// SIMATIC S7-200 SMART project (STEP 7-Micro/WIN SMART), CPU SR40

SYMBOL_TABLE 表格 1
Stage1_Temp_CT   C0       // 阶段升温一计数器，分钟计数
Stage2_Temp_CT   C1       // 阶段升温二计数器，分钟计数
Stage3_Temp_CT   C2       // 阶段升温三计数器，分钟计数
Stage4_Temp_CT   C3       // 阶段升温四计数器，分钟计数
Stage5_Temp_CT   C4       // 阶段升温五计数器，分钟计数
Stage6_Temp_CT   C5       // 阶段升温六计数器，分钟计数
Sys_Time_Minutes_CNT C100     // 系统运行时长计数器，分钟
Sys_Time_Hours_CNT C101     // 系统运行时长计数器，小时
Sys_Time_Repeat_CNT C102     // 系统运行时长轮数计数器，超过32767小时后，该轮数加1，小时归0
C_Leak_CountDown_CT C103     // 检漏倒计时 计数器
C_Valve_Detect_CT C104     // 调节阀检测倒计时 计数器
C_Purge_CountDown_CT C105     // 吹扫倒计时 计数器
C_Ignite_CountDown_CT C106     // 点火 倒计时 计数器
MBUS_INIT_DONE   M0.1     // MBUS_INIT的Done 状态位
MBUS_SLAVE_DONE  M0.2     // MBUS_SLAVE Done状态位
M_Safety_Check_FLG M0.3     // 系统安全回路检测 标志，如压力、检漏、前火检等
M_Valve_ALM_FLG  M0.4     // 调节阀检测故障标志
M_Local_Remote_FLG M0.5     // 本地远程标志，1本地，0远程
M_Auto_Temp_FLG  M0.6     // 自动升温控制标志
M_Purge_Display_FLG M0.7     // 显示吹扫动画
M_SYS_Safety_Pass_FLG M1.0     // 安全自检通过标志：检漏通过、空气压力正常、燃气压力正常，前火检正常
M_Sys_Run_FLG    M1.1     // 启动标志
M_Purge_Begin_FLG M1.2     // 开始吹扫标志
M_Ignite_Begin_FLG M1.3     // 开始点火标志
M_Ignite_Success_FLG M1.4     // 点火成功标志
M_OverTemp_FLG   M1.5     // 超温标志
M_Purge_Finish_FLG M1.6     // 吹扫结束标志
M_Ignite_Ready_FLG M1.7     // 点火准备标志
M_SYS_Alarm_FLG  M2.0     // 系统故障标志
M_Ignite_BeginTime_FLG M2.1     // 点火延时开始
M_Temp1_Read_FLG M2.2     // 读阶段1温度标志
M_Temp2_Read_FLG M2.3     // 读阶段2温度标志
M_Temp3_Read_FLG M2.4     // 读阶段3温度标志
M_Temp4_Read_FLG M2.5     // 读阶段4温度标志
M_Temp5_Read_FLG M2.6     // 读阶段5温度标志
M_Temp6_Read_FLG M2.7     // 读阶段6温度标志
M_Valve_Pass_FLG M3.0     // 调节阀检测通过标志
M_Leak_Exception_FLG M3.1     // 检漏异常报警
M_Leak_Pass_FLG  M3.4     // 检漏程序，检漏通过
M_Run_Big_Fire_FLG M3.5     // 大火指示，表示大火正常燃烧
M_TA_Spark_FLG   M3.7     // 变压器打火标志
M_Temp_Error_FLG M4.0     // 温度错误，DCS传送温度数据有误，请
M_Valve_Ignite_OPEN_FLG M4.1     // 点火阀开启标志
M_Sys_Detect_PASS_FLG M4.2     // 系统预检通过标志
Local_Start_CMD  M10.0    // 本地启动指令
Local_Stop_CMD   M10.1    // 本地停止指令
Local_Reset_CMD  M10.2    // 本地复位指令
Remote_Start_CMD M10.3    // 远程启动指令
Remote_Stop_CMD  M10.4    // 远程停止指令
Remote_Reset_CMD M10.5    // 远程复位指令
M_Manu_TurnUp_CMD M10.6    // 手动升档，触摸屏虚拟按钮
M_Manu_TurnDown_CMD M10.7    // 手动降档，触摸屏虚拟按钮
M_Auto_Manu_CMD  M11.0    // 自动/手动切换，触摸屏虚拟按钮，1自动，0手动
M_Leak_ValveCut_CMD M11.1    // 检漏程序，打开主火阀（切断阀）指令
M_ValveCut_CMD   M11.2    // 主程序，打开主火阀（切断阀）
M_Leak_ValveSafety_CMD M11.3    // 检漏程序，打开安全阀 指令
M_ValveSafety_CMD M11.4    // 主程序，打开安全阀 指令
Remote_TurnUP_CMD M11.5    // 远程升档指令
Remote_TurnDown_CMD M11.6    // 远程降档指令
Local_TurnUP_CMD M11.7    // 本地升档指令
Local_TurnDown_CMD M12.0    // 本地降档指令
M_Leak_Start_CMD M12.1    // 手动检漏 虚拟按钮
M_Valve_Detect_CMD M12.2    // 手动调节阀检测 虚拟按钮
M_Ignite_Failed_ALM M20.0    // 点火失败报警
M_Flame_Loss_ALM M20.1    // 火焰信号丢失
M_DCS_Lock_ALM   M20.2    // DCS安全联锁故障
M_Air_Pres_Low_ALM M20.3    // 空气压力低故障
M_Gas_Pres_High_ALM M20.4    // 燃气压力高故障
M_Gas_Pres_Low_ALM M20.5    // 燃气压力低故障
M_Flame_Pre_ALM  M20.6    // 点火前发现火焰故障
M_Leak_Exception2_ALM M20.7    // 检漏程序，第2步检漏异常标志
M_Leak_Exception4_ALM M21.0    // 检漏程序，第4步检漏异常标志
M_Valve_Air_ALM  M21.1    // 空气调节阀故障
M_Valve_Gas_ALM  M21.2    // 燃气调节阀故障
T_Purge_Duration T101     // 吹扫时长定时器
T_Ignite_Delay   T102     // 点火延时定时器，从调节阀走到位到高压包放电之间的时间间隔
T_Level_Interval T103     // 升降档间隔定时器
T_Flame_Loss_Delay T104     // 火焰丢失延时定时器
T_VAL_Open_Delay T105     // 大火阀开启延时定时器
T_TA_Spark_Time  T106     // 高压包打火时长定时器
T_Valve_Ignite_Delay T107     // 母火阀延时打开定时器
T_Leak_Step1_Delay T110     // 检漏第1步延时定时器
T_Leak_Step2_Delay T111     // 检漏第2步延时定时器
T_Leak_Step3_Delay T112     // 检漏第3步延时定时器
T_Leak_Step4_Delay T113     // 检漏第4步延时定时器
T_Valve_Control_Detect T115     // 调节阀检测定时器
T_Ignite_ValveGo_Delay T116     // 点火位置，调节阀走至点火位置延时
T_Flame_Pre_Detect T118     // 前火焰检测延时定时器
T_Purge_ValveOpenDelay T119     // 吹扫 调节阀开启延时定时器
T_Flame_Build_Delay T120     // 火焰建立延时定时器
T_Leak_Total_Time T121     // 检漏总时长定时器
I_DCS_Abandon    V0.0     // I_DCS安全联锁，不用
I_Air_Pres_Low_STS V0.1     // 空气压力低故障
I_Gas_Pres_High_STS V0.2     // 燃气压力高故障
I_Gas_Pres_Low_STS V0.3     // 燃气压力低故障
I_JES258_Alrm_Abandon V0.4     // I_JES258故障不用
I_Flame_STS      V0.5     // 火焰信号
I_Run_STS        V0.6     // 启动按钮信号
I_Stop_STS       V0.7     // 停止按钮信号
I_Reset_STS      V1.0     // 复位按钮信号
I_LocalRemote_STS V1.1     // 本地、远程信号。1本地、0远程
Q_Sys_Alarm      V2.0     // 系统报警输出指令，蜂鸣器
Q_Valve_Ignite   V2.1     // 点火阀Ignite打开命令
Q_Valve_Cut      V2.2     // 主火切断阀打开命令
Q_TA_Spark       V2.3     // 变压器打火指令
Q_SYS_Flame_Light V2.4     // 有火指示灯
Q_SYS_Run_Light  V2.5     // 运行指示灯
Q_SYS_Stop_Light V2.6     // 停止指示灯
Q_Valve_Safety   V2.7     // 安全阀打开命令
V_Remote_Alarm_Status V1620.0  // 故障状态RTU
V_Remote_Auto_Status V1620.1  // 自动状态RTU
V_Remote_Run_Status V1620.2  // 启动状态RTU
V_Remote_Stop_Status V1620.3  // 停止状态RTU
V_Local_Remote_Status V1620.4  // 本地远程状态RTU
V_Remote_Run_CMD V1620.5  // 远程启动RTU
V_Remote_Stop_CMD V1620.6  // 远程停止RTU
V_Remote_Reset_CMD V1620.7  // 远程复位RTU
V_Remote_TurnUp_CMD V1621.0  // 远程升档RTU
V_Remote_TurnDown_CMD V1621.1  // 远程降档RTU
V_PID_ErrorCode  VB800    // PID 控制错误码
V_MBUS_INIT_Error VB802    // MBUS_INIT Error 错误码
V_MBUS_SLAVE_Error VB804    // MBUS_SLAVE Error 错误码
B_Leak_Step_Num  VB806    // 检漏步数，第1、2、3、4步
B_Leak_Status    VB808    // 检漏状态，0:停止检漏 1:检漏中 2:检漏完成
B_ValveLift_Status VB810    // 调节阀检测状态，0停止检测、1检测中、2检测完成
B_Ignate_Backup_Status VB812    // 0正常；1点火备用，取消前火检
DI_Current_Temp_VAL VD20     // 当前温度（长整型）数据来自DCS
R_Current_Temp_Display VD24     // 温度HMI显示值
R_ValveLift_Gas_VAL_Per VD32     // 燃气阀门开度显示%
R_ValveLift_Air_VAL_Per VD36     // 空气阀门开度显示%
R_Valve_Gas_DIFF_ABS VD40     // 燃气阀门给定值与反馈值之差，取绝对值
R_Valve_Air_DIFF_ABS VD44     // 空气阀门给定值与反馈值之差，取绝对值
R_ValveLift_Gas_VAL VD48     // 当前燃气给定值
R_ValveLift_Air_VAL VD52     // 当前空气给定值
R_PID_Temp_VAL   VD56     // PID当前目标温度
R_PID_Manu_VAL   VD60     // PID手动值
R_Purge_BeginTime_VAL VD64     // 吹扫计时开始_值
R_PID_Level_Round_VAL VD68     // PID输出换算成档位，四舍五入后
R_Current_Level_VAL VD72     // 当前档位值
R_PID_EachLevel_VAL VD76     // 当量_每档
R_PID_Output_VAL VD80     // 转换为实数后的PID输出值
R_PID_Level_VAL  VD84     // PID输出换算成档位
R_Current_Temp_VAL VD88     // 当前温度（实数）数据来自DCS
R_Valve_Gas_DIFF_VAL VD92     // 燃气阀门给定值与反馈值之差
R_Valve_Air_DIFF_VAL VD96     // 空气阀门给定值与反馈值之差
DI_ValveLift_Air_Per VD148    // 空气调节阀 双整型 %
DI_ValveLift_Gas_Per VD156    // 燃气调节阀 双整型 %
R_Temp_Upper_Limit_SET VD300    // 温度上限设定值
R_Temp_Lower_Limit_SET VD304    // 温度下限设定值
R_Over_Temp_Stop_SET VD308    // 超温停机设定值
R_Gas_DiffAlow_SET VD312    // 燃气偏差允许值设定
R_Air_DiffAlow_SET VD316    // 空气偏差允许值设定
R_Purge_Valve_Air_SET VD320    // 吹扫空气阀开度设定值
R_PID_D_SET      VD324    // PID微分_D 设定值
R_PID_P_SET      VD328    // PID增益_P 设定值
R_PID_I_SET      VD332    // PID积分_I 设定值
R_PID_Ts_SET     VD336    // PID采样时间设定值
R_Level_Total_SET VD340    // 档位设置
R_Gas_Level_Stop_SET VD344    // 燃气停机档设定值
R_Gas_Level_Ignite_SET VD348    // 燃气点火档设定值
R_Gas_Level1_SET VD352    // 燃气1档设定值
R_Gas_Level2_SET VD356    // 燃气2档设定值
R_Gas_Level3_SET VD360    // 燃气3档设定值
R_Gas_Level4_SET VD364    // 燃气4档设定值
R_Gas_Level5_SET VD368    // 燃气5档设定值
R_Gas_Level6_SET VD372    // 燃气6档设定值
R_Gas_Level7_SET VD376    // 燃气7档设定值
R_Gas_Level8_SET VD380    // 燃气8档设定值
R_Gas_Level9_SET VD384    // 燃气9档设定值
R_Gas_Level10_SET VD388    // 燃气10档设定值
R_Gas_Level11_SET VD392    // 燃气11档设定值
R_Gas_Level12_SET VD396    // 燃气12档设定值
R_Gas_Level13_SET VD400    // 燃气13档设定值
R_Gas_Level14_SET VD404    // 燃气14档设定值
R_Gas_Level15_SET VD408    // 燃气15档设定值
R_Gas_Level16_SET VD412    // 燃气16档设定值
R_Gas_Level17_SET VD416    // 燃气17档设定值
R_Gas_Level18_SET VD420    // 燃气18档设定值
R_Air_Level_Stop_SET VD424    // 空气停机档设定值
R_Air_Level_Ignite_SET VD428    // 空气点火档设定值
R_Air_Level1_SET VD432    // 空气1档设定值
R_Air_Level2_SET VD436    // 空气2档设定值
R_Air_Level3_SET VD440    // 空气3档设定值
R_Air_Level4_SET VD444    // 空气4档设定值
R_Air_Level5_SET VD448    // 空气5档设定值
R_Air_Level6_SET VD452    // 空气6档设定值
R_Air_Level7_SET VD456    // 空气7档设定值
R_Air_Level8_SET VD460    // 空气8档设定值
R_Air_Level9_SET VD464    // 空气9档设定值
R_Air_Level10_SET VD468    // 空气10档设定值
R_Air_Level11_SET VD472    // 空气11档设定值
R_Air_Level12_SET VD476    // 空气12档设定值
R_Air_Level13_SET VD480    // 空气13档设定值
R_Air_Level14_SET VD484    // 空气14档设定值
R_Air_Level15_SET VD488    // 空气15档设定值
R_Air_Level16_SET VD492    // 空气16档设定值
R_Air_Level17_SET VD496    // 空气17档设定值
R_Air_Level18_SET VD500    // 空气18档设定值
R_Stage1_Temp_SET VD504    // 阶段1温度设定值
R_Stage2_Temp_SET VD508    // 阶段2温度设定值
R_Stage3_Temp_SET VD512    // 阶段3温度设定值
R_Stage4_Temp_SET VD516    // 阶段4温度设定值
R_Stage5_Temp_SET VD520    // 阶段5温度设定值
R_Stage6_Temp_SET VD524    // 阶段6温度设定值
R_Remote_AirLift_VAL VD640    // 远程显示空气阀开度
R_Remote_GasLift_VAL VD644    // 远程显示燃气阀开度
R_Remote_Temp_VAL VD648    // 远程显示温度
R_Remote_Air_VAL VD1640   // 空气调节阀开度RTU
R_Remote_Gas_VAL VD1644   // 燃气调节阀开度RTU
R_Remote_Level_VAL VD1652   // 当前档位RTU
R_Remote_Temp_SET VD1880   // 目标温度RTU
W_Purge_Time_VAL VW100    // 当前吹扫时长显示值
W_PID_Output_VAL VW104    // PID输出
W_Stage1_Temp_Time_VAL VW108    // 第1阶段温度保持时长显示，分钟
W_Stage2_Temp_Time_VAL VW112    // 第2阶段温度保持时长显示，分钟
W_Stage3_Temp_Time_VAL VW116    // 第3阶段温度保持时长显示，分钟
W_Stage4_Temp_Time_VAL VW120    // 第4阶段温度保持时长显示，分钟
W_Stage5_Temp_Time_VAL VW124    // 第5阶段温度保持时长显示，分钟
W_Stage6_Temp_Time_VAL VW128    // 第6阶段温度保持时长显示，分钟
W_Sys_Time_Hour_VAL VW132    // HMI显示运行小时
W_Sys_Time_Minute_VAL VW136    // HMI显示运行分钟
W_Valve_Detect_CD_VAL VW138    // 调节阀检测倒计时 计算值
W_Leak_CD_VAL    VW140    // 检漏倒计时 计算值
W_Purge_CD_VAL   VW142    // 吹扫倒计时 计算值
W_Ignite_CD_VAL  VW144    // 高压打火 倒计时 计算值
W_ValveLift_Air_VAL_Per VW152    // 空气调节阀开度 整数 %
W_ValveLift_Gas_VAL_Per VW158    // 燃气调节阀开度 整数 %
W_Purge_Time_SET VW528    // 吹扫时间设定
W_Ignite_Delay_SET VW532    // 点火延时设定值
W_ValveCut_Delay_SET VW536    // 主火阀(切断阀)开启延时设定值
W_Stage1_Temp_Time_SET VW540    // 第1阶段温度时长设定值，小时
W_Stage2_Temp_Time_SET VW544    // 第2阶段温度时长设定值，小时
W_Stage3_Temp_Time_SET VW548    // 第3阶段温度时长设定值，小时
W_Stage4_Temp_Time_SET VW552    // 第4阶段温度时长设定值，小时
W_Stage5_Temp_Time_SET VW556    // 第5阶段温度时长设定值，小时
W_Stage6_Temp_Time_SET VW560    // 第6阶段温度时长设定值，小时
W_PreFlame_Time_SET VW564    // 前火检时长设定值
W_Ignite_Spark_Time_SET VW568    // 高压包打火时长设定值
W_Valve_Ignite_Time_SET VW572    // 点火阀开启延时设定值
W_ValveDetect_Time_SET VW576    // 调节阀检测时长设定值
W_Flame_Build_Time_SET VW580    // 火焰建立延时时长设定值
W_Flame_Loss_Time_SET VW584    // 火焰丢失延时时长设定值，建议1~3秒
W_Sys_Status     VW814    // 1.检漏、调节阀检测中…… / 2.检测完成 / 3.设备停止 / 4.正在启动…… / 5.正在吹扫…… / 6.吹扫完成 / 7.点火准备中…… / 8.正在点火…… / 9.点火成功 / 10.【小火运行】 / 11.【大火运行】 / 12.故障报警
W_Sys_Status_Time VW816    // 系统状态时间
W_Remote_Temp_VAL VW1898   // 当前温度RTU
W_Remote_Air_P_VAL VW1918   // 当前管道空气压力，风压
END_SYMBOL_TABLE

SYMBOL_TABLE 系统符号
Always_On        SM0.0    // 始终接通
First_Scan_On    SM0.1    // 仅在第一个扫描周期时接通
Clock_60s        SM0.4    // 针对 1 分钟的周期时间，时钟脉冲接通 30 s，断开 30 s.
Clock_1s         SM0.5    // 针对 1 s 的周期时间，时钟脉冲接通 0.5 s，断开 0.5 s.
END_SYMBOL_TABLE

ORGANIZATION_BLOCK 程序块:OB1
TITLE=程序注释
BEGIN
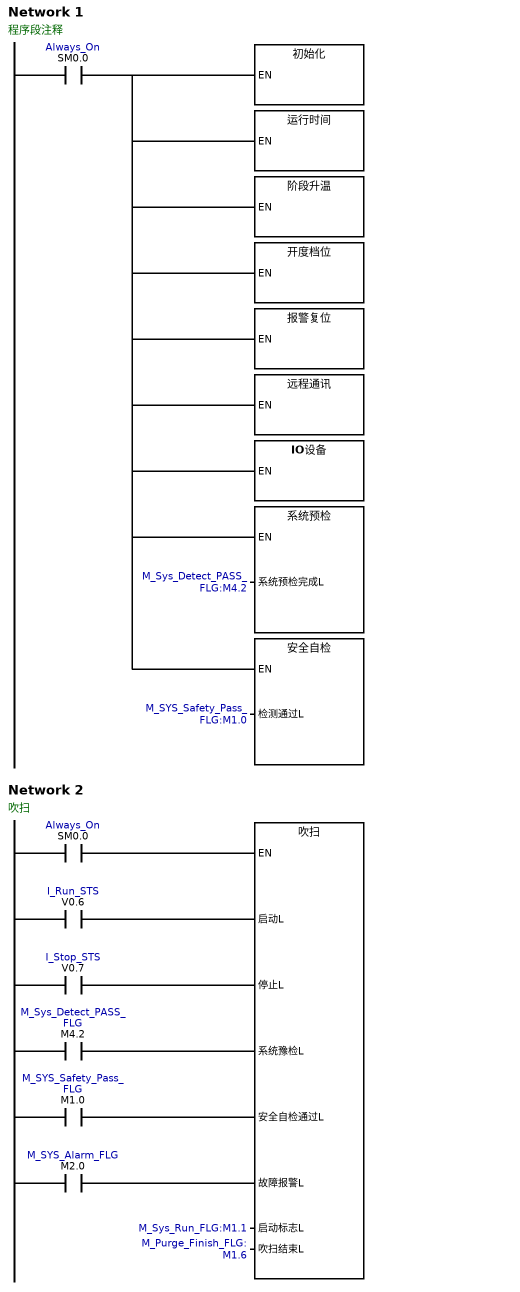
Network 1
// 程序段注释
LD     Always_On:SM0.0
CALL   初始化:SBR0
CALL   运行时间:SBR9
CALL   阶段升温:SBR5
CALL   开度档位:SBR6
CALL   报警复位:SBR13
CALL   远程通讯:SBR7
CALL   IO设备:SBR8
CALL   系统预检:SBR1, M_Sys_Detect_PASS_FLG:M4.2
CALL   安全自检:SBR2, M_SYS_Safety_Pass_FLG:M1.0
Network 2
// 吹扫
LD     Always_On:SM0.0
=      L60.0
LD     I_Run_STS:V0.6
=      L63.7
LD     I_Stop_STS:V0.7
=      L63.6
LD     M_Sys_Detect_PASS_FLG:M4.2
=      L63.5
LD     M_SYS_Safety_Pass_FLG:M1.0
=      L63.4
LD     M_SYS_Alarm_FLG:M2.0
=      L63.3
LD     L60.0
CALL   吹扫:SBR3, L63.7, L63.6, L63.5, L63.4, L63.3, M_Sys_Run_FLG:M1.1, M_Purge_Finish_FLG:M1.6
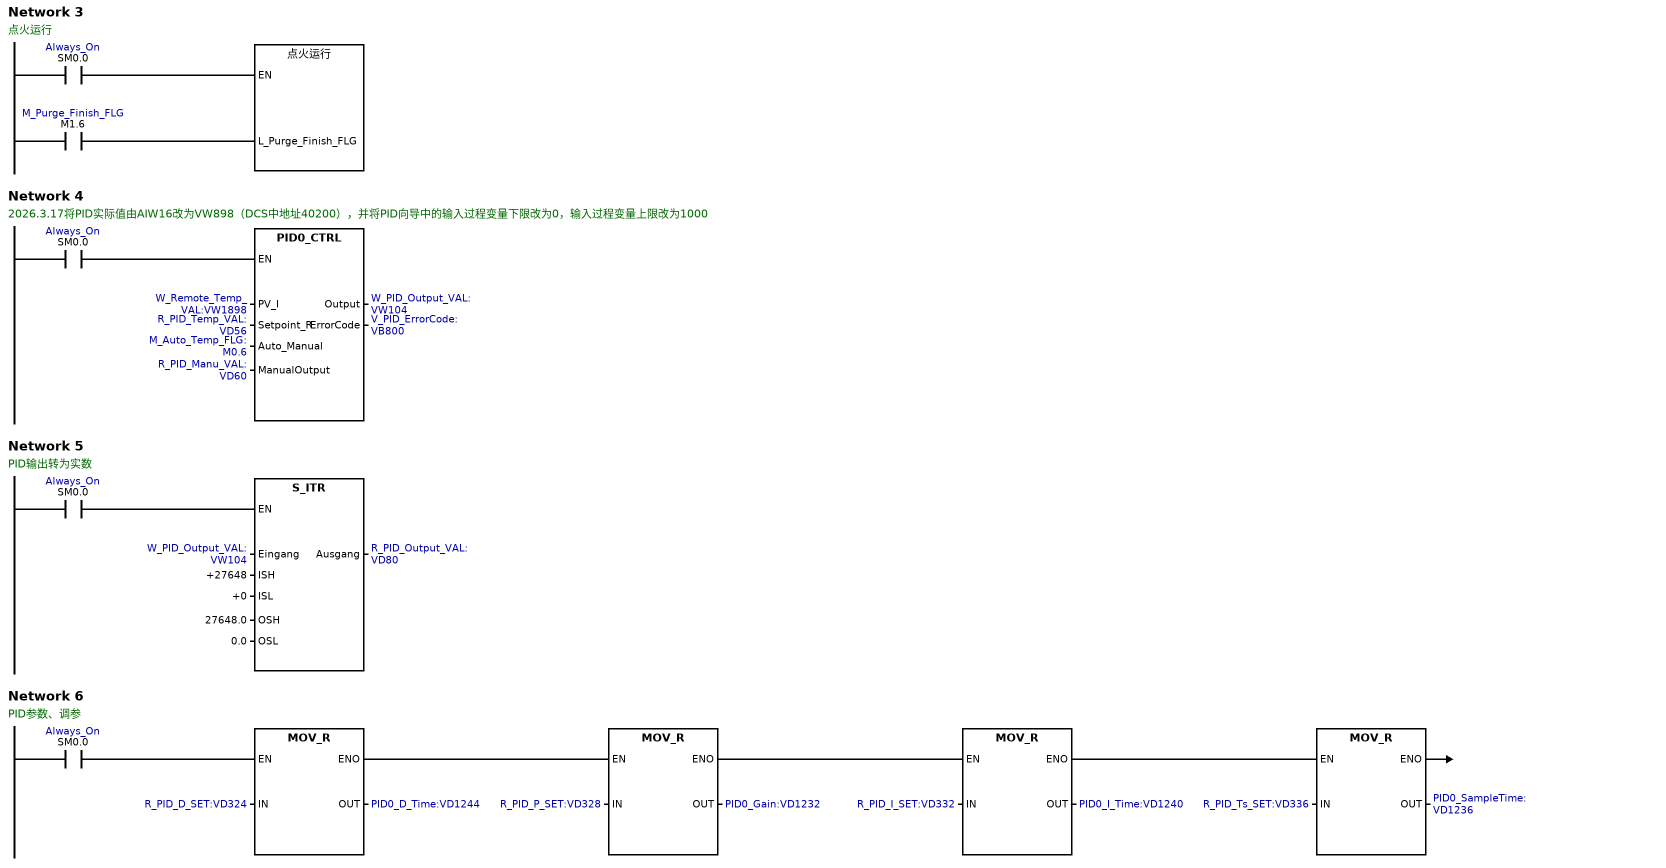
Network 3
// 点火运行
LD     Always_On:SM0.0
=      L60.0
LD     M_Purge_Finish_FLG:M1.6
=      L63.7
LD     L60.0
CALL   点火运行:SBR4, L63.7
Network 4
// 2026.3.17将PID实际值由AIW16改为VW898（DCS中地址40200），并将PID向导中的输入过程变量下限改为0，输入过程变量上限改为1000
LD     Always_On:SM0.0
CALL   PID0_CTRL:SBR18, W_Remote_Temp_VAL:VW1898, R_PID_Temp_VAL:VD56, M_Auto_Temp_FLG:M0.6, R_PID_Manu_VAL:VD60, W_PID_Output_VAL:VW104, V_PID_ErrorCode:VB800
Network 5
// PID输出转为实数
LD     Always_On:SM0.0
CALL   S_ITR:SBR30, W_PID_Output_VAL:VW104, +27648, +0, 27648.0, 0.0, R_PID_Output_VAL:VD80
Network 6
// PID参数、调参
LD     Always_On:SM0.0
MOVR   R_PID_D_SET:VD324, PID0_D_Time:VD1244
AENO
MOVR   R_PID_P_SET:VD328, PID0_Gain:VD1232
AENO
MOVR   R_PID_I_SET:VD332, PID0_I_Time:VD1240
AENO
MOVR   R_PID_Ts_SET:VD336, PID0_SampleTime:VD1236
END_ORGANIZATION_BLOCK

SUBROUTINE_BLOCK 初始化:SBR0
TITLE=初始化子程序
// 功能：数据初始化
// 1、本地/远程转换
// 2、PID自动/手动转换
// 3、PLC IO 输入输出映射
// 4、数据初始化
// 5、本地/远程 命令封装
// 6、模拟量处理
// 
// 
BEGIN
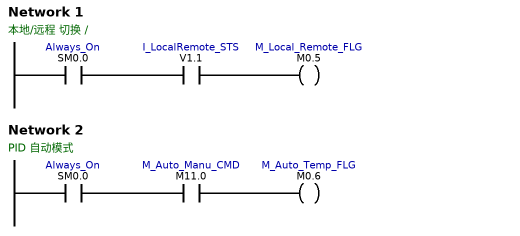
Network 1
// 本地/远程 切换
// 
LD     Always_On:SM0.0
A      I_LocalRemote_STS:V1.1
=      M_Local_Remote_FLG:M0.5
Network 2
// PID 自动模式 
LD     Always_On:SM0.0
A      M_Auto_Manu_CMD:M11.0
=      M_Auto_Temp_FLG:M0.6
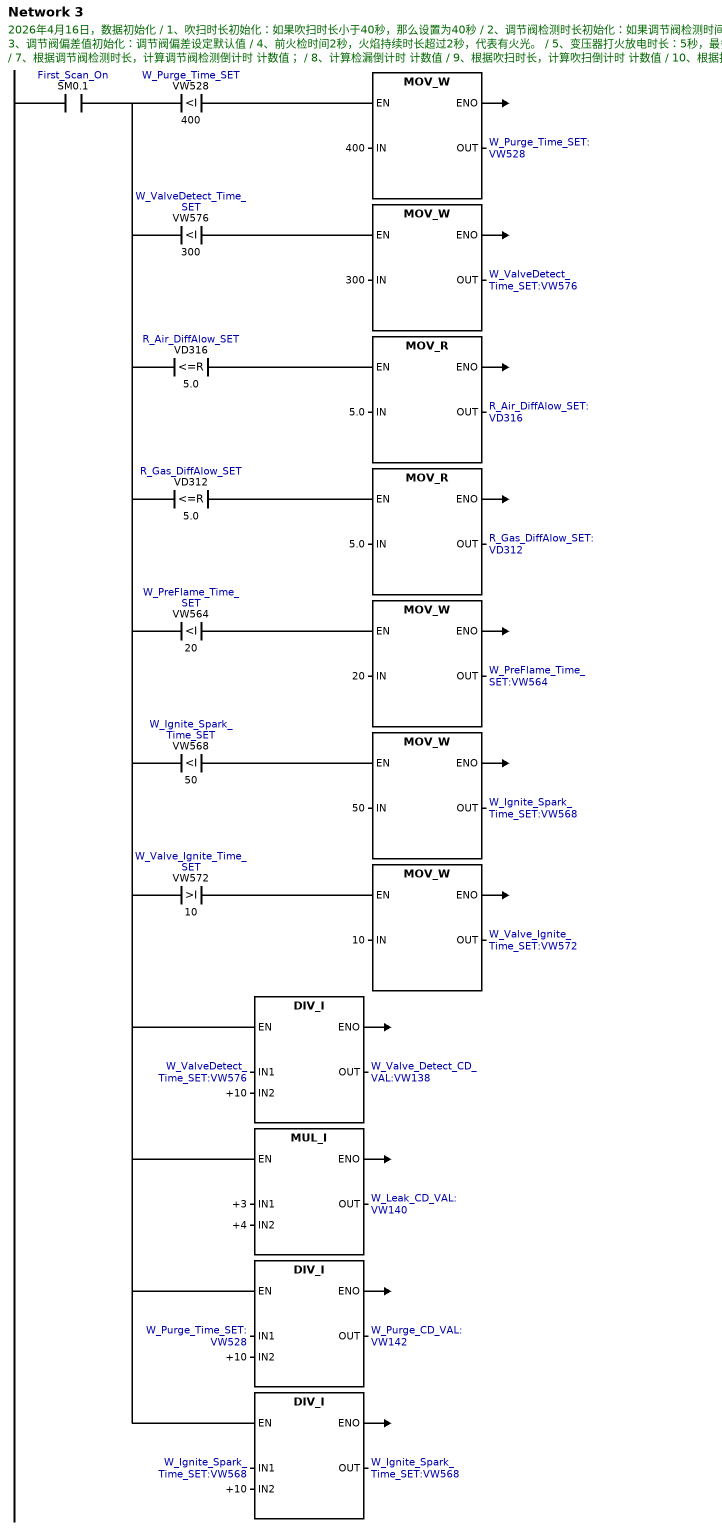
Network 3
// 2026年4月16日，数据初始化
// 1、吹扫时长初始化：如果吹扫时长小于40秒，那么设置为40秒
// 2、调节阀检测时长初始化：如果调节阀检测时间小于30秒，那么设置为30秒
// 3、调节阀偏差值初始化：调节阀偏差设定默认值
// 4、前火检时间2秒，火焰持续时长超过2秒，代表有火光。
// 5、变压器打火放电时长：5秒，最多7秒，大于7秒，那么 就设置为7秒
// 6、点火阀延时开启时长：1秒，最多2秒
// 7、根据调节阀检测时长，计算调节阀检测倒计时 计数值；
// 8、计算检漏倒计时 计数值
// 9、根据吹扫时长，计算吹扫倒计时 计数值
// 10、根据打火时长，计算打火倒计时 计数值
LD     First_Scan_On:SM0.1
LPS
AW<    W_Purge_Time_SET:VW528, 400
MOVW   400, W_Purge_Time_SET:VW528
LRD
AW<    W_ValveDetect_Time_SET:VW576, 300
MOVW   300, W_ValveDetect_Time_SET:VW576
LRD
AR<=   R_Air_DiffAlow_SET:VD316, 5.0
MOVR   5.0, R_Air_DiffAlow_SET:VD316
LRD
AR<=   R_Gas_DiffAlow_SET:VD312, 5.0
MOVR   5.0, R_Gas_DiffAlow_SET:VD312
LRD
AW<    W_PreFlame_Time_SET:VW564, 20
MOVW   20, W_PreFlame_Time_SET:VW564
LRD
AW<    W_Ignite_Spark_Time_SET:VW568, 50
MOVW   50, W_Ignite_Spark_Time_SET:VW568
LRD
AW>    W_Valve_Ignite_Time_SET:VW572, 10
MOVW   10, W_Valve_Ignite_Time_SET:VW572
LRD
MOVW   W_ValveDetect_Time_SET:VW576, W_Valve_Detect_CD_VAL:VW138
/I     +10, W_Valve_Detect_CD_VAL:VW138
LRD
MOVW   +3, W_Leak_CD_VAL:VW140
*I     +4, W_Leak_CD_VAL:VW140
LRD
MOVW   W_Purge_Time_SET:VW528, W_Purge_CD_VAL:VW142
/I     +10, W_Purge_CD_VAL:VW142
LPP
/I     +10, W_Ignite_Spark_Time_SET:VW568
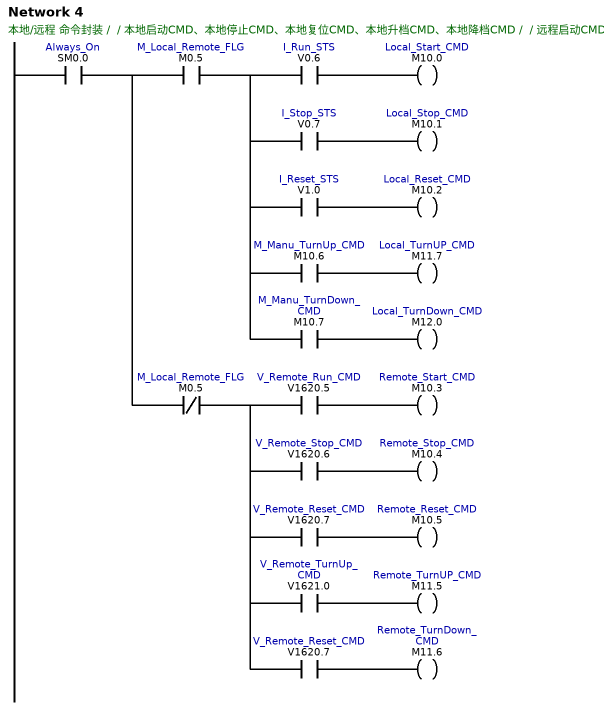
Network 4
// 本地/远程 命令封装
// 
// 本地启动CMD、本地停止CMD、本地复位CMD、本地升档CMD、本地降档CMD
// 
// 远程启动CMD、远程停止CMD、远程复位CMD、远程升档CMD、远程降档CMD
LD     Always_On:SM0.0
LPS
A      M_Local_Remote_FLG:M0.5
LPS
A      I_Run_STS:V0.6
=      Local_Start_CMD:M10.0
LRD
A      I_Stop_STS:V0.7
=      Local_Stop_CMD:M10.1
LRD
A      I_Reset_STS:V1.0
=      Local_Reset_CMD:M10.2
LRD
A      M_Manu_TurnUp_CMD:M10.6
=      Local_TurnUP_CMD:M11.7
LPP
A      M_Manu_TurnDown_CMD:M10.7
=      Local_TurnDown_CMD:M12.0
LPP
AN     M_Local_Remote_FLG:M0.5
LPS
A      V_Remote_Run_CMD:V1620.5
=      Remote_Start_CMD:M10.3
LRD
A      V_Remote_Stop_CMD:V1620.6
=      Remote_Stop_CMD:M10.4
LRD
A      V_Remote_Reset_CMD:V1620.7
=      Remote_Reset_CMD:M10.5
LRD
A      V_Remote_TurnUp_CMD:V1621.0
=      Remote_TurnUP_CMD:M11.5
LPP
A      V_Remote_Reset_CMD:V1620.7
=      Remote_TurnDown_CMD:M11.6
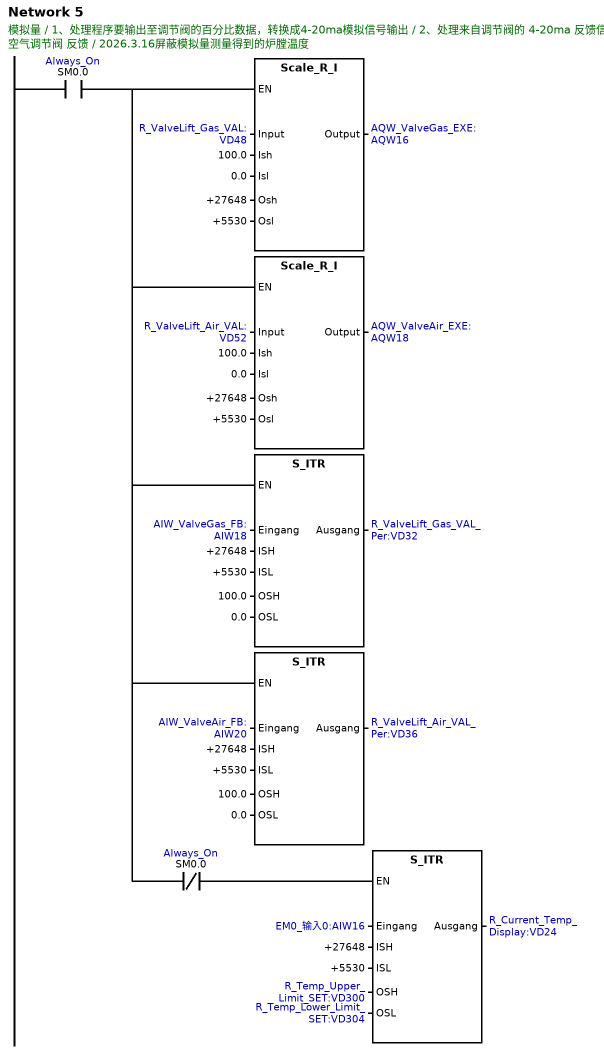
Network 5
// 模拟量
// 1、处理程序要输出至调节阀的百分比数据，转换成4-20ma模拟信号输出
// 2、处理来自调节阀的 4-20ma 反馈信号，转换成百分比数据；
// 
// 燃气调节阀 执行输出
// 空气调节阀 执行输出
// 燃气调节阀  反馈
// 空气调节阀 反馈
// 2026.3.16屏蔽模拟量测量得到的炉膛温度
LD     Always_On:SM0.0
CALL   Scale_R_I:SBR24, R_ValveLift_Gas_VAL:VD48, 100.0, 0.0, +27648, +5530, AQW_ValveGas_EXE:AQW16
CALL   Scale_R_I:SBR24, R_ValveLift_Air_VAL:VD52, 100.0, 0.0, +27648, +5530, AQW_ValveAir_EXE:AQW18
CALL   S_ITR:SBR30, AIW_ValveGas_FB:AIW18, +27648, +5530, 100.0, 0.0, R_ValveLift_Gas_VAL_Per:VD32
CALL   S_ITR:SBR30, AIW_ValveAir_FB:AIW20, +27648, +5530, 100.0, 0.0, R_ValveLift_Air_VAL_Per:VD36
AN     Always_On:SM0.0
CALL   S_ITR:SBR30, EM0_输入0:AIW16, +27648, +5530, R_Temp_Upper_Limit_SET:VD300, R_Temp_Lower_Limit_SET:VD304, R_Current_Temp_Display:VD24
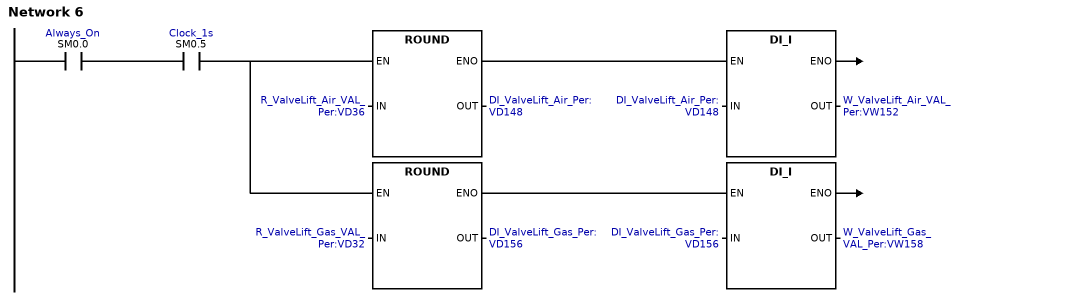
Network 6
LD     Always_On:SM0.0
A      Clock_1s:SM0.5
LPS
ROUND  R_ValveLift_Air_VAL_Per:VD36, DI_ValveLift_Air_Per:VD148
AENO
DTI    DI_ValveLift_Air_Per:VD148, W_ValveLift_Air_VAL_Per:VW152
LPP
ROUND  R_ValveLift_Gas_VAL_Per:VD32, DI_ValveLift_Gas_Per:VD156
AENO
DTI    DI_ValveLift_Gas_Per:VD156, W_ValveLift_Gas_VAL_Per:VW158
Network 7
// 检漏程序
END_SUBROUTINE_BLOCK

SUBROUTINE_BLOCK 系统预检:SBR1
TITLE=系统预检子程序说明
// 本程序块包含两个功能：
// 1、检漏，用来检测阀组是否有泄漏，在PLC上电时，进行一次检漏，通过，则PLC在下次断电不再进行检漏。
// 	检漏说明：阀组包括燃气进所测阀为安全阀V1，烧嘴侧阀为主火阀V2。V1阀、V2阀之间的腔体装有燃气低压开关，用来检测腔体的压力。
// 	检漏步骤：
// 	1、打开主火阀V2 保持3秒，然后关闭V2阀，等待3秒；
// 	2、检测V1阀、V2阀 之间的燃气压力，此时应检测不到燃气压力（因第1步已经把气放完）。如果检测到，说明前面的安全阀（V1）泄漏。
// 	3、打开安全阀V1，保持3秒后关闭，等待3秒
// 	4、检测V1、V2之间的压力，此时应该检测到压力，如果没有检测到，说明烧嘴侧阀泄漏。
// 	
// 
// 2、调节阀检测功能，在PLC上电时进行一次调节阀功能好坏检测，通过以后在PLC下次断电再上电前不再进行检测。
// 
VAR_IN_OUT
系统预检完成L:BOOL;	// L0.0 
END_VAR
BEGIN
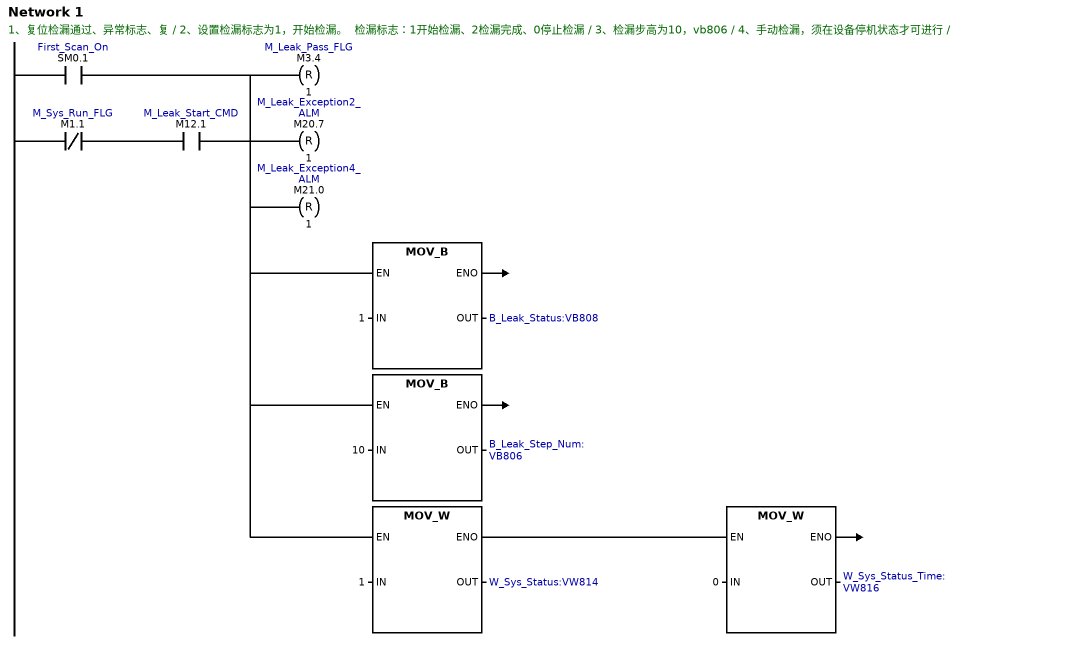
Network 1
// 1、复位检漏通过、异常标志、复
// 2、设置检漏标志为1，开始检漏。	检漏标志：1开始检漏、2检漏完成、0停止检漏
// 3、检漏步高为10，vb806
// 4、手动检漏，须在设备停机状态才可进行
// 
LD     First_Scan_On:SM0.1
LDN    M_Sys_Run_FLG:M1.1
A      M_Leak_Start_CMD:M12.1
OLD
R      M_Leak_Pass_FLG:M3.4, 1
R      M_Leak_Exception2_ALM:M20.7, 1
R      M_Leak_Exception4_ALM:M21.0, 1
MOVB   1, B_Leak_Status:VB808
MOVB   10, B_Leak_Step_Num:VB806
MOVW   1, W_Sys_Status:VW814
AENO
MOVW   0, W_Sys_Status_Time:VW816
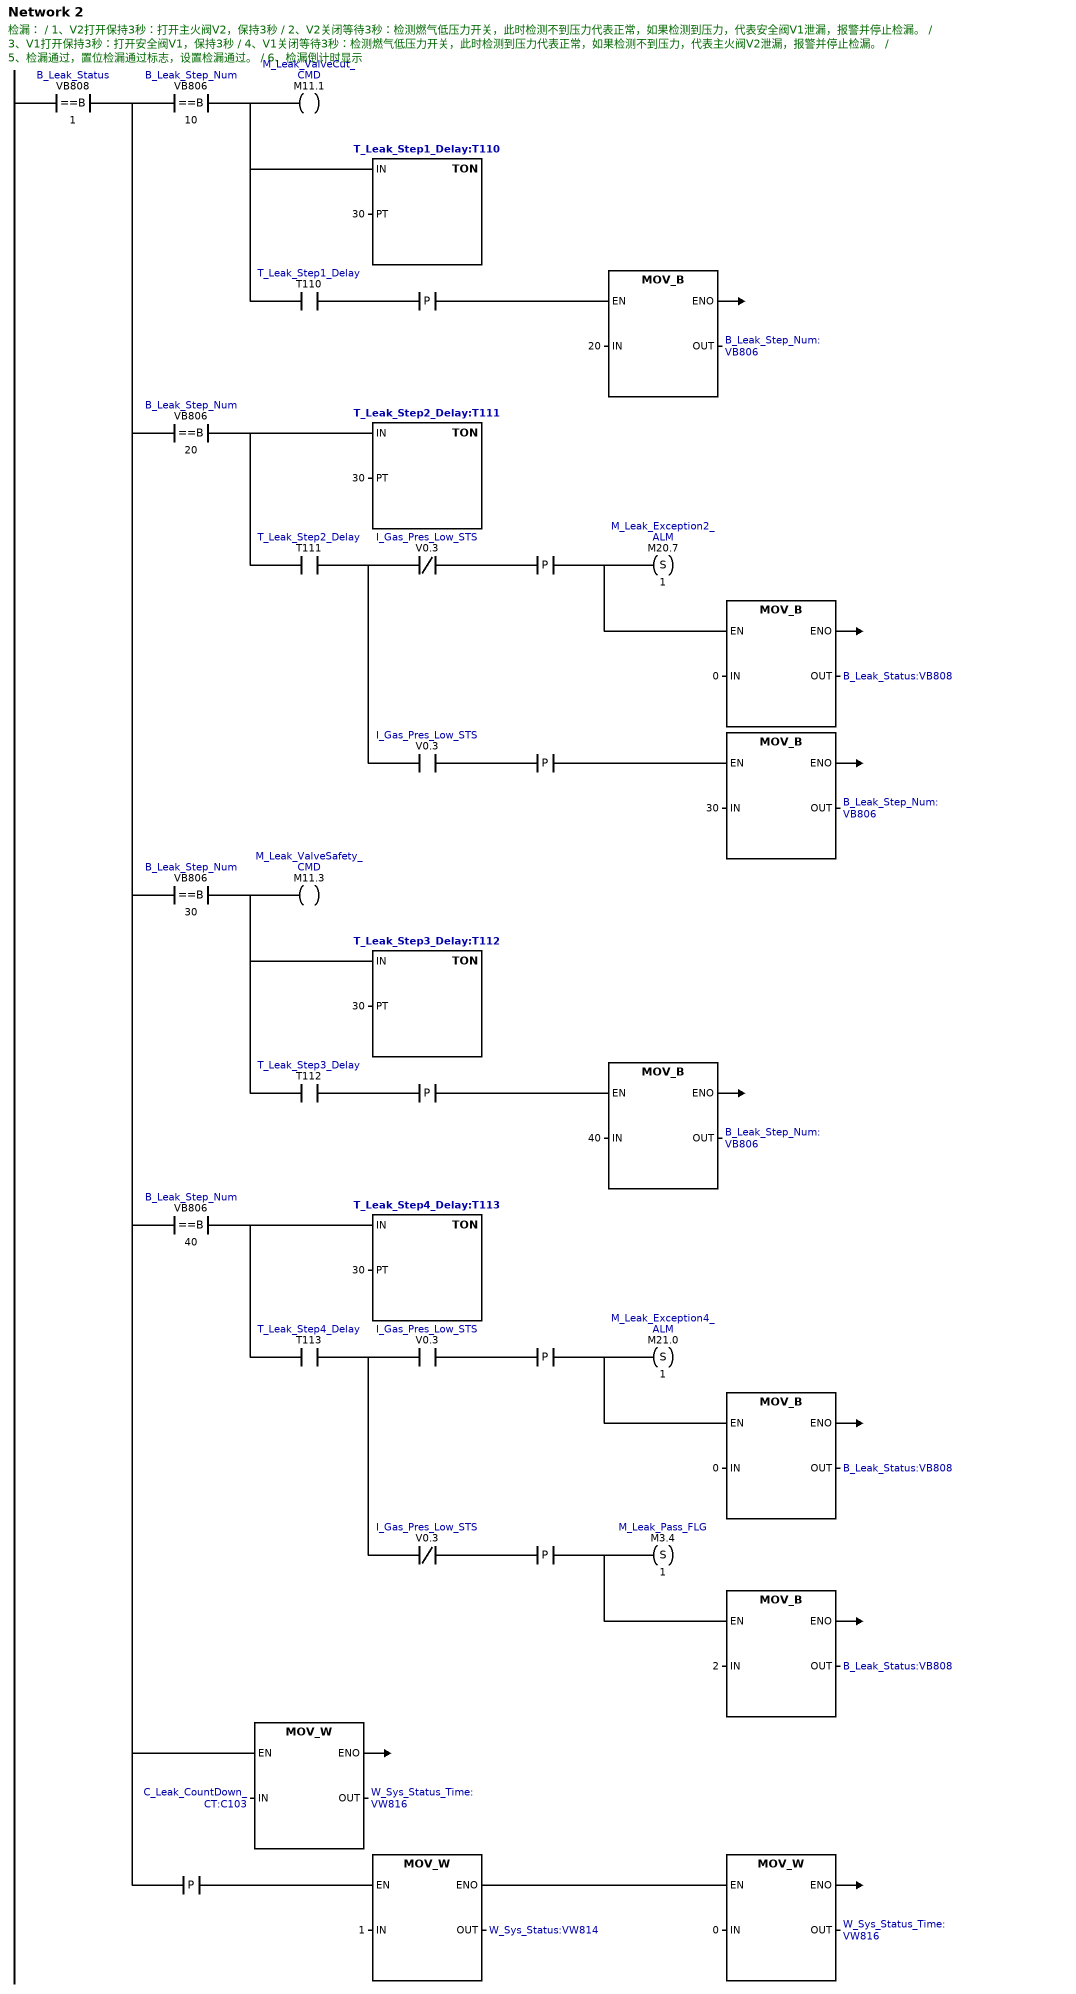
Network 2
// 检漏：
// 1、V2打开保持3秒：打开主火阀V2，保持3秒
// 2、V2关闭等待3秒：检测燃气低压力开关，此时检测不到压力代表正常，如果检测到压力，代表安全阀V1泄漏，报警并停止检漏。
// 3、V1打开保持3秒：打开安全阀V1，保持3秒
// 4、V1关闭等待3秒：检测燃气低压力开关，此时检测到压力代表正常，如果检测不到压力，代表主火阀V2泄漏，报警并停止检漏。
// 5、检漏通过，置位检漏通过标志，设置检漏通过。
// 6、检漏倒计时显示
LDB=   B_Leak_Status:VB808, 1
LPS
AB=    B_Leak_Step_Num:VB806, 10
=      M_Leak_ValveCut_CMD:M11.1
TON    T_Leak_Step1_Delay:T110, 30
A      T_Leak_Step1_Delay:T110
EU
MOVB   20, B_Leak_Step_Num:VB806
LRD
AB=    B_Leak_Step_Num:VB806, 20
TON    T_Leak_Step2_Delay:T111, 30
A      T_Leak_Step2_Delay:T111
LPS
AN     I_Gas_Pres_Low_STS:V0.3
EU
S      M_Leak_Exception2_ALM:M20.7, 1
MOVB   0, B_Leak_Status:VB808
LPP
A      I_Gas_Pres_Low_STS:V0.3
EU
MOVB   30, B_Leak_Step_Num:VB806
LRD
AB=    B_Leak_Step_Num:VB806, 30
=      M_Leak_ValveSafety_CMD:M11.3
TON    T_Leak_Step3_Delay:T112, 30
A      T_Leak_Step3_Delay:T112
EU
MOVB   40, B_Leak_Step_Num:VB806
LRD
AB=    B_Leak_Step_Num:VB806, 40
TON    T_Leak_Step4_Delay:T113, 30
A      T_Leak_Step4_Delay:T113
LPS
A      I_Gas_Pres_Low_STS:V0.3
EU
S      M_Leak_Exception4_ALM:M21.0, 1
MOVB   0, B_Leak_Status:VB808
LPP
AN     I_Gas_Pres_Low_STS:V0.3
EU
S      M_Leak_Pass_FLG:M3.4, 1
MOVB   2, B_Leak_Status:VB808
LPP
MOVW   C_Leak_CountDown_CT:C103, W_Sys_Status_Time:VW816
EU
MOVW   1, W_Sys_Status:VW814
AENO
MOVW   0, W_Sys_Status_Time:VW816
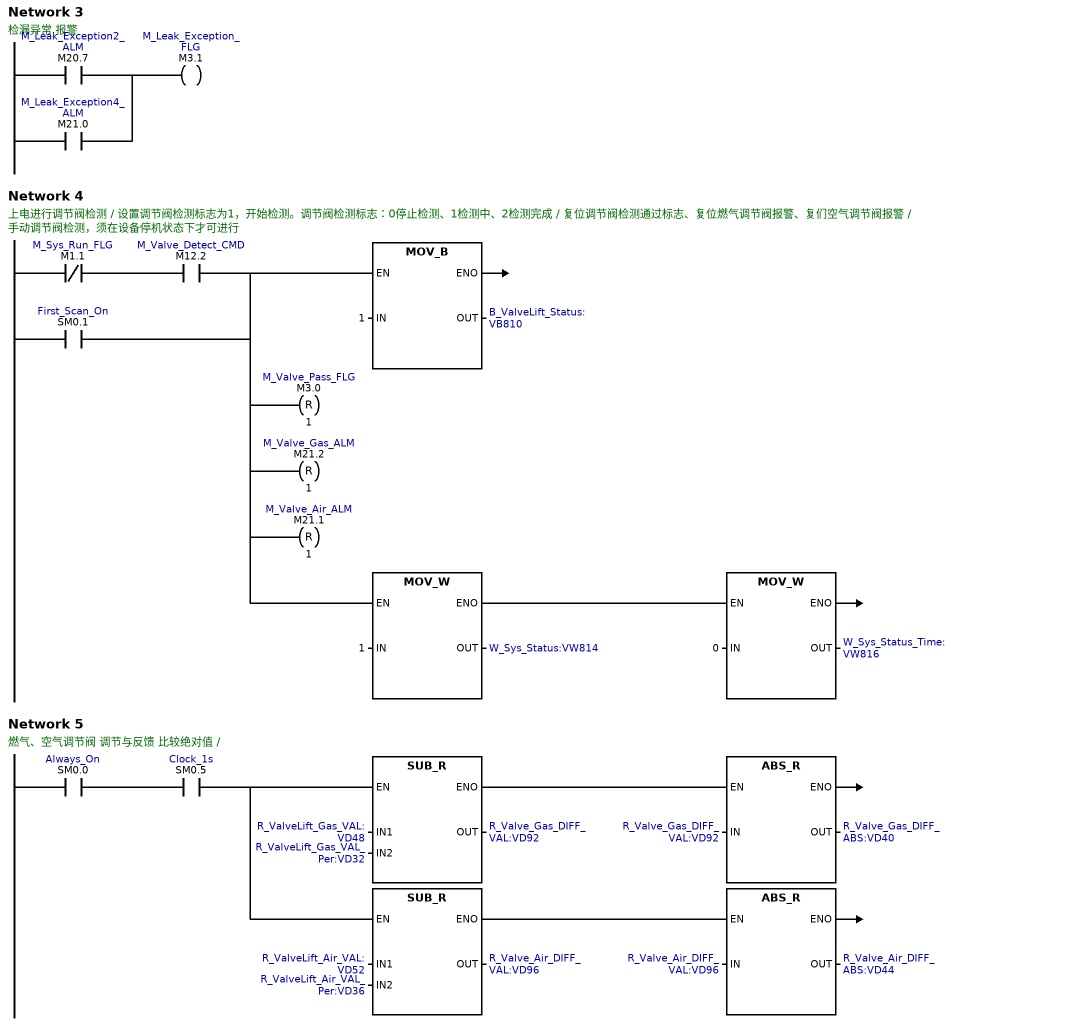
Network 3
// 检漏异常 报警
LD     M_Leak_Exception2_ALM:M20.7
O      M_Leak_Exception4_ALM:M21.0
=      M_Leak_Exception_FLG:M3.1
Network 4
// 上电进行调节阀检测
// 设置调节阀检测标志为1，开始检测。调节阀检测标志：0停止检测、1检测中、2检测完成
// 复位调节阀检测通过标志、复位燃气调节阀报警、复们空气调节阀报警
// 手动调节阀检测，须在设备停机状态下才可进行
LDN    M_Sys_Run_FLG:M1.1
A      M_Valve_Detect_CMD:M12.2
O      First_Scan_On:SM0.1
MOVB   1, B_ValveLift_Status:VB810
R      M_Valve_Pass_FLG:M3.0, 1
R      M_Valve_Gas_ALM:M21.2, 1
R      M_Valve_Air_ALM:M21.1, 1
MOVW   1, W_Sys_Status:VW814
AENO
MOVW   0, W_Sys_Status_Time:VW816
Network 5
// 燃气、空气调节阀 调节与反馈 比较绝对值
// 
LD     Always_On:SM0.0
A      Clock_1s:SM0.5
LPS
MOVR   R_ValveLift_Gas_VAL:VD48, R_Valve_Gas_DIFF_VAL:VD92
AENO
-R     R_ValveLift_Gas_VAL_Per:VD32, R_Valve_Gas_DIFF_VAL:VD92
AENO
ABSR   R_Valve_Gas_DIFF_VAL:VD92, R_Valve_Gas_DIFF_ABS:VD40
LPP
MOVR   R_ValveLift_Air_VAL:VD52, R_Valve_Air_DIFF_VAL:VD96
AENO
-R     R_ValveLift_Air_VAL_Per:VD36, R_Valve_Air_DIFF_VAL:VD96
AENO
ABSR   R_Valve_Air_DIFF_VAL:VD96, R_Valve_Air_DIFF_ABS:VD44
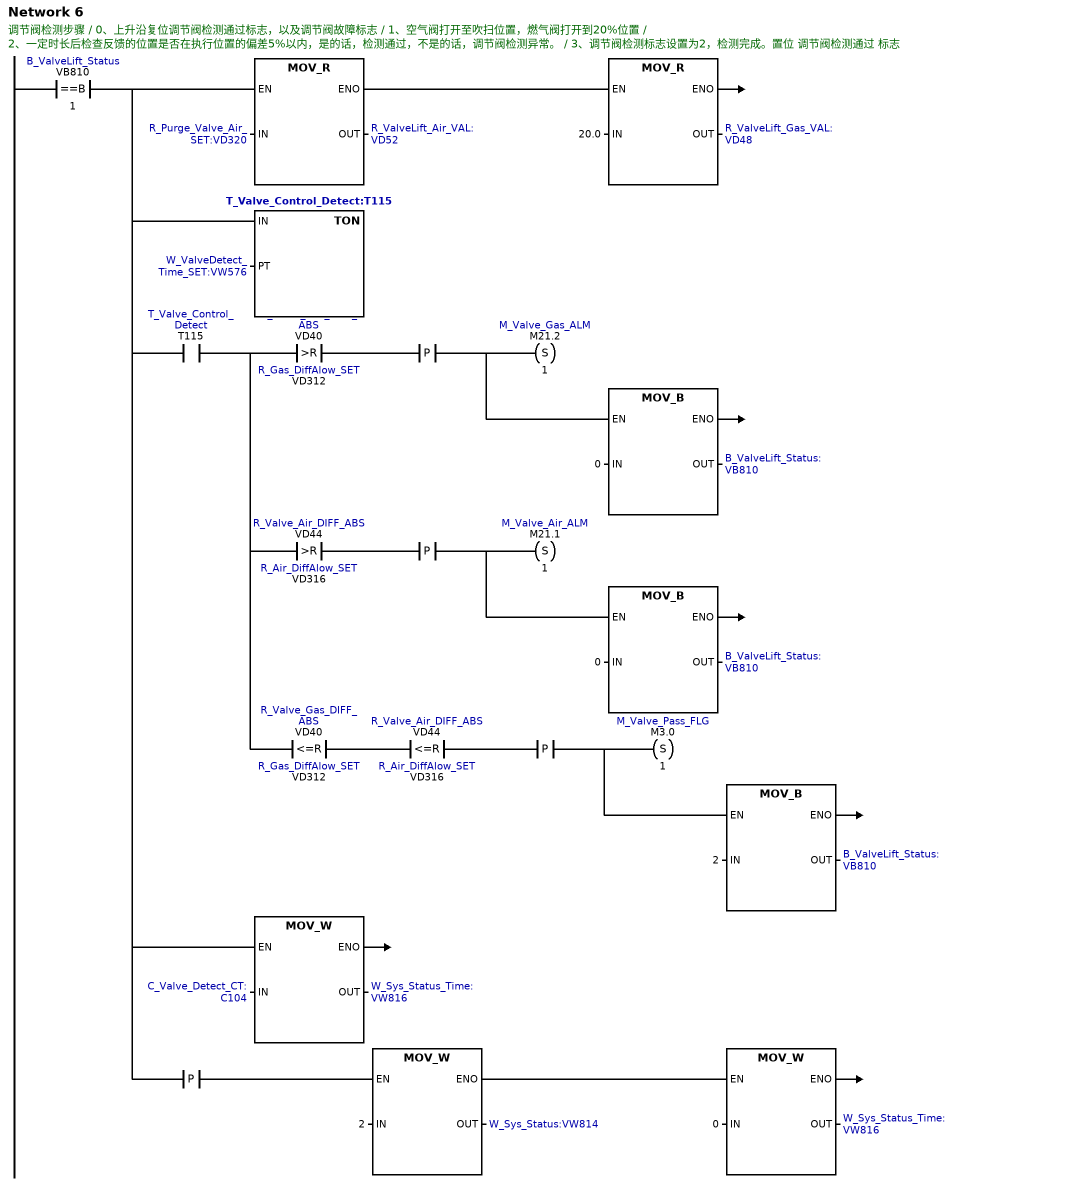
Network 6
// 调节阀检测步骤
// 0、上升沿复位调节阀检测通过标志，以及调节阀故障标志
// 1、空气阀打开至吹扫位置，燃气阀打开到20%位置
// 2、一定时长后检查反馈的位置是否在执行位置的偏差5%以内，是的话，检测通过，不是的话，调节阀检测异常。
// 3、调节阀检测标志设置为2，检测完成。置位 调节阀检测通过 标志
LDB=   B_ValveLift_Status:VB810, 1
LPS
MOVR   R_Purge_Valve_Air_SET:VD320, R_ValveLift_Air_VAL:VD52
AENO
MOVR   20.0, R_ValveLift_Gas_VAL:VD48
LRD
TON    T_Valve_Control_Detect:T115, W_ValveDetect_Time_SET:VW576
LRD
A      T_Valve_Control_Detect:T115
LPS
AR>    R_Valve_Gas_DIFF_ABS:VD40, R_Gas_DiffAlow_SET:VD312
EU
S      M_Valve_Gas_ALM:M21.2, 1
MOVB   0, B_ValveLift_Status:VB810
LRD
AR>    R_Valve_Air_DIFF_ABS:VD44, R_Air_DiffAlow_SET:VD316
EU
S      M_Valve_Air_ALM:M21.1, 1
MOVB   0, B_ValveLift_Status:VB810
LPP
AR<=   R_Valve_Gas_DIFF_ABS:VD40, R_Gas_DiffAlow_SET:VD312
AR<=   R_Valve_Air_DIFF_ABS:VD44, R_Air_DiffAlow_SET:VD316
EU
S      M_Valve_Pass_FLG:M3.0, 1
MOVB   2, B_ValveLift_Status:VB810
LPP
MOVW   C_Valve_Detect_CT:C104, W_Sys_Status_Time:VW816
EU
MOVW   2, W_Sys_Status:VW814
AENO
MOVW   0, W_Sys_Status_Time:VW816
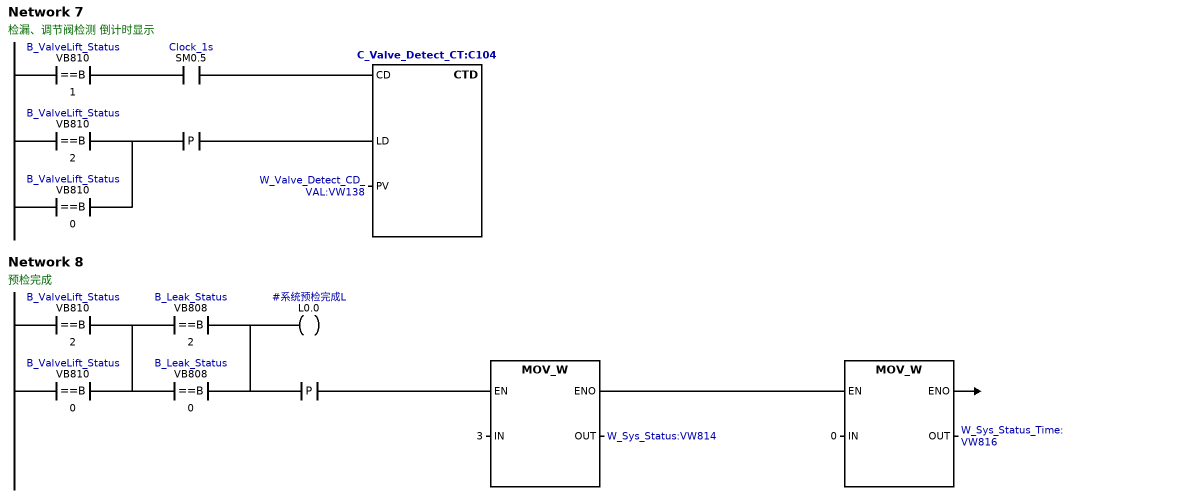
Network 7
// 检漏、调节阀检测 倒计时显示
LDB=   B_ValveLift_Status:VB810, 1
A      Clock_1s:SM0.5
LDB=   B_ValveLift_Status:VB810, 2
OB=    B_ValveLift_Status:VB810, 0
EU
CTD    C_Valve_Detect_CT:C104, W_Valve_Detect_CD_VAL:VW138
Network 8
// 预检完成
LDB=   B_ValveLift_Status:VB810, 2
OB=    B_ValveLift_Status:VB810, 0
LDB=   B_Leak_Status:VB808, 2
OB=    B_Leak_Status:VB808, 0
ALD
=      #系统预检完成L:L0.0
EU
MOVW   3, W_Sys_Status:VW814
AENO
MOVW   0, W_Sys_Status_Time:VW816
END_SUBROUTINE_BLOCK

SUBROUTINE_BLOCK 安全自检:SBR2
TITLE=安全自检 子程序说明
// 
// 本子程序主要用来进行系统安全检测，有以下几点：
// 1、前火检，烧嘴还未进行点火之前，炉膛内部不应该有火焰，如果检测到火焰报警。增加点火备用标志，置位点火备用，不再进行前火检。
// 2、空气压力低报警，如果风压达不到，报警。
// 3、燃气压力高报警，燃气压力如果超过要求上限，报警
// 4、燃气压力低报警，燃气压力如果达不到要求，报警。
// 
// 特别说明：检漏完成（检漏状态码B_Leak_Status 值为2）燃气压力低检测才生效
// 
// 检测通过之后，置位检测通过标志
VAR_IN_OUT
检测通过L:BOOL;	// L0.0 
END_VAR
BEGIN
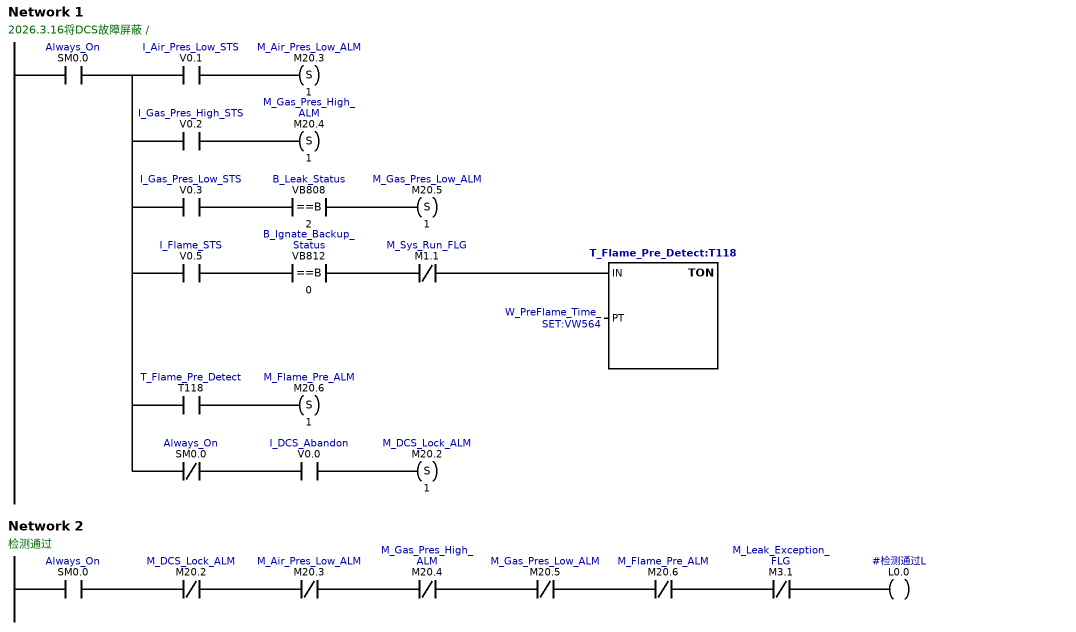
Network 1
// 2026.3.16将DCS故障屏蔽
// 
LD     Always_On:SM0.0
LPS
A      I_Air_Pres_Low_STS:V0.1
S      M_Air_Pres_Low_ALM:M20.3, 1
LRD
A      I_Gas_Pres_High_STS:V0.2
S      M_Gas_Pres_High_ALM:M20.4, 1
LRD
A      I_Gas_Pres_Low_STS:V0.3
AB=    B_Leak_Status:VB808, 2
S      M_Gas_Pres_Low_ALM:M20.5, 1
LRD
A      I_Flame_STS:V0.5
AB=    B_Ignate_Backup_Status:VB812, 0
AN     M_Sys_Run_FLG:M1.1
TON    T_Flame_Pre_Detect:T118, W_PreFlame_Time_SET:VW564
LRD
A      T_Flame_Pre_Detect:T118
S      M_Flame_Pre_ALM:M20.6, 1
LPP
AN     Always_On:SM0.0
A      I_DCS_Abandon:V0.0
S      M_DCS_Lock_ALM:M20.2, 1
Network 2
// 检测通过
LD     Always_On:SM0.0
AN     M_DCS_Lock_ALM:M20.2
AN     M_Air_Pres_Low_ALM:M20.3
AN     M_Gas_Pres_High_ALM:M20.4
AN     M_Gas_Pres_Low_ALM:M20.5
AN     M_Flame_Pre_ALM:M20.6
AN     M_Leak_Exception_FLG:M3.1
=      #检测通过L:L0.0
END_SUBROUTINE_BLOCK

SUBROUTINE_BLOCK 吹扫:SBR3
TITLE=吹扫子程序
// 一、预吹扫
// 功能：向炉膛内部送入大量新鲜空气，将可能残存或积聚的可燃气体、未完全燃烧的煤粉等可燃物彻底排出，防止爆炸，确保点火安全；
// 1、空气调节阀 打开至 吹扫 设定位置，如果空气调节阀故障，那么等待调节阀检测时间长后开始吹扫。
// 2、吹扫计时 
// 3、吹扫完成，档位设置为点火档，点火档为0.5（空气2档、燃气2档）
// 
// 
// 二、后吹扫：冷却与清洁（可选）
// 这是在燃烧器停止工作或熄火后进行的程序。
// 清除残留： 继续通入空气，清除燃烧产生的副产物和残留的未燃气体，防止其在设备内积聚。
// 保护设备： 帮助冷却热交换器等高温部件，同时减少积碳和腐蚀性气体对设备的损害，从而延长燃烧器的使用寿命。
VAR_INPUT
启动L:BOOL;	// L0.0 
停止L:BOOL;	// L0.1 
系统豫检L:BOOL;	// L0.2 
安全自检通过L:BOOL;	// L0.3 
故障报警L:BOOL;	// L0.4 
END_VAR
VAR_IN_OUT
启动标志L:BOOL;	// L0.5 
吹扫结束L:BOOL;	// L0.6 
END_VAR
BEGIN
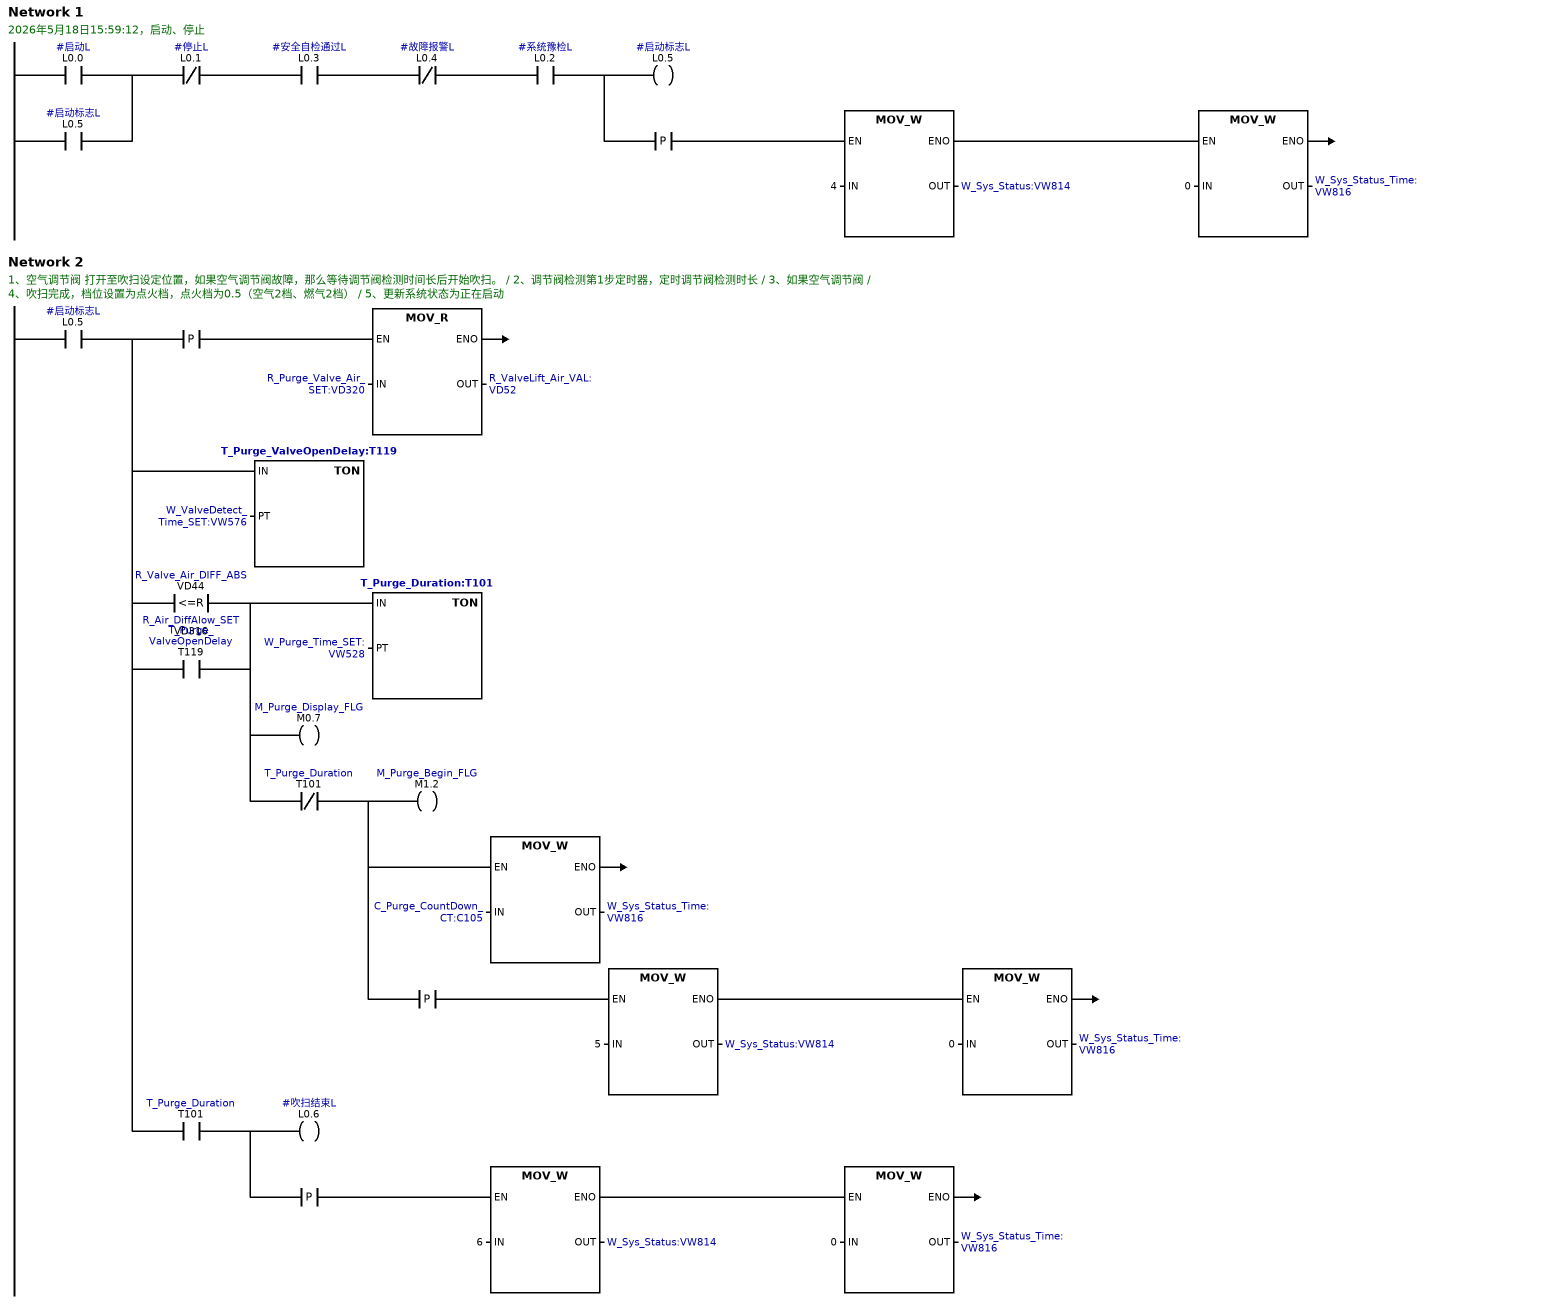
Network 1
// 2026年5月18日15:59:12，启动、停止
LD     #启动L:L0.0
O      #启动标志L:L0.5
AN     #停止L:L0.1
A      #安全自检通过L:L0.3
AN     #故障报警L:L0.4
A      #系统豫检L:L0.2
=      #启动标志L:L0.5
EU
MOVW   4, W_Sys_Status:VW814
AENO
MOVW   0, W_Sys_Status_Time:VW816
Network 2
// 1、空气调节阀 打开至吹扫设定位置，如果空气调节阀故障，那么等待调节阀检测时间长后开始吹扫。
// 2、调节阀检测第1步定时器，定时调节阀检测时长
// 3、如果空气调节阀
// 4、吹扫完成，档位设置为点火档，点火档为0.5（空气2档、燃气2档）
// 5、更新系统状态为正在启动
LD     #启动标志L:L0.5
LPS
EU
MOVR   R_Purge_Valve_Air_SET:VD320, R_ValveLift_Air_VAL:VD52
LRD
TON    T_Purge_ValveOpenDelay:T119, W_ValveDetect_Time_SET:VW576
LRD
LDR<=  R_Valve_Air_DIFF_ABS:VD44, R_Air_DiffAlow_SET:VD316
O      T_Purge_ValveOpenDelay:T119
ALD
TON    T_Purge_Duration:T101, W_Purge_Time_SET:VW528
=      M_Purge_Display_FLG:M0.7
AN     T_Purge_Duration:T101
=      M_Purge_Begin_FLG:M1.2
MOVW   C_Purge_CountDown_CT:C105, W_Sys_Status_Time:VW816
EU
MOVW   5, W_Sys_Status:VW814
AENO
MOVW   0, W_Sys_Status_Time:VW816
LPP
A      T_Purge_Duration:T101
=      #吹扫结束L:L0.6
EU
MOVW   6, W_Sys_Status:VW814
AENO
MOVW   0, W_Sys_Status_Time:VW816
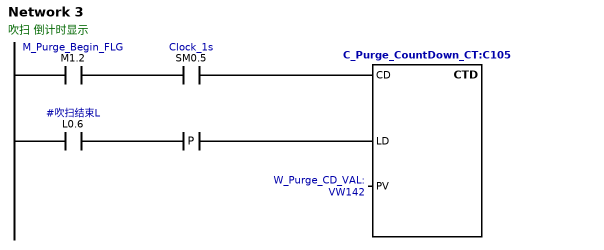
Network 3
// 吹扫 倒计时显示
LD     M_Purge_Begin_FLG:M1.2
A      Clock_1s:SM0.5
LD     #吹扫结束L:L0.6
EU
CTD    C_Purge_CountDown_CT:C105, W_Purge_CD_VAL:VW142
END_SUBROUTINE_BLOCK

SUBROUTINE_BLOCK 点火运行:SBR4
TITLE=点火运行子程序
// 功能：
// 一、点火，控制设备安全点火
// 二、正常运行，控制设备安全、稳定运行
// 三、手动模式，手动调节负荷大小；自动模式，根据温度PID调节负荷。
// 四、超温停机处理程序
// 
// 1. 点火信号触发
// 点火变压器输出产生持续电火花（点火时间 2~5 秒）。
// 必须遵循 火等气 原则：先确认电火花稳定存在，再通入燃料。
// 
// 2. 燃料释放与火焰建立
// 点火电极工作 3 秒后，开启 点火阀（小火阀），通入少量燃料
// 关键安全窗口：火焰检测器必须在 2 秒内 确认稳定火焰信号。若超时未检测到火焰：立即关闭燃料阀，自动触发重新预吹扫，禁止二次直接点火。
// 
// 3. 点火成功判定
// 火焰信号持续 ≥3 秒 且无波动，判定点火成功，进入下一阶段。
// 点火失败处理：立即关闭燃料阀，重新执行 ≥15 分钟预吹扫。
// 人工排查原因（燃料压力不足、电极积碳、风燃比失调等）。
// 
// 
// 4、延时一段时间后，开主火阀
// 
// 5、火焰丢失报警：火焰丢失报警触发逻辑
// 
// 步骤1：信号丢失确认
// 火焰检测器连续 1~3秒 未检测到有效火焰信号（具体阈值由安全标准设定）。
// 示例：燃气燃烧器通常设为 1秒，燃油燃烧器因火焰稳定性稍差可放宽至 2~3秒。
// 
// 步骤2：联锁动作触发
// 立即关闭燃料安全切断阀（响应时间 ≤1秒）。
// 同步启动后吹扫程序（持续 ≥15秒），清除残留可燃气体。
// 声光报警：控制面板显示故障代码，并锁定系统。
// 
// 步骤3：人工干预要求
// 系统进入 安全锁定状态，未经人工复位禁止自动重启。
// 必须排查熄火原因（如燃料压力波动、风量过大、探头污染）后才能复位。
// 
// 6、超温停机（待写）
// 
// 
VAR_INPUT
L_Purge_Finish_FLG:BOOL;	// L0.0 
END_VAR
BEGIN
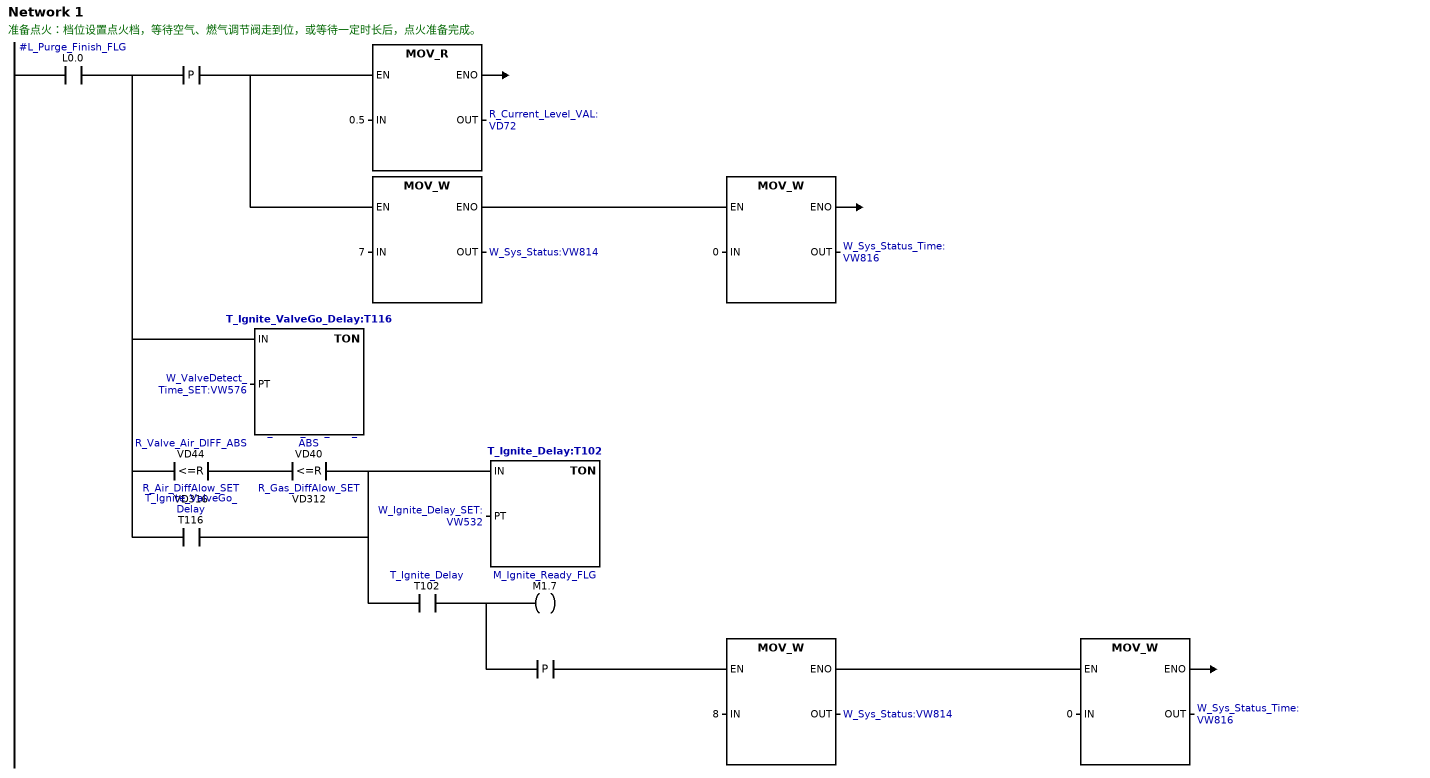
Network 1
// 准备点火：档位设置点火档，等待空气、燃气调节阀走到位，或等待一定时长后，点火准备完成。
LD     #L_Purge_Finish_FLG:L0.0
LPS
EU
MOVR   0.5, R_Current_Level_VAL:VD72
MOVW   7, W_Sys_Status:VW814
AENO
MOVW   0, W_Sys_Status_Time:VW816
LRD
TON    T_Ignite_ValveGo_Delay:T116, W_ValveDetect_Time_SET:VW576
LPP
LDR<=  R_Valve_Air_DIFF_ABS:VD44, R_Air_DiffAlow_SET:VD316
AR<=   R_Valve_Gas_DIFF_ABS:VD40, R_Gas_DiffAlow_SET:VD312
O      T_Ignite_ValveGo_Delay:T116
ALD
TON    T_Ignite_Delay:T102, W_Ignite_Delay_SET:VW532
A      T_Ignite_Delay:T102
=      M_Ignite_Ready_FLG:M1.7
EU
MOVW   8, W_Sys_Status:VW814
AENO
MOVW   0, W_Sys_Status_Time:VW816
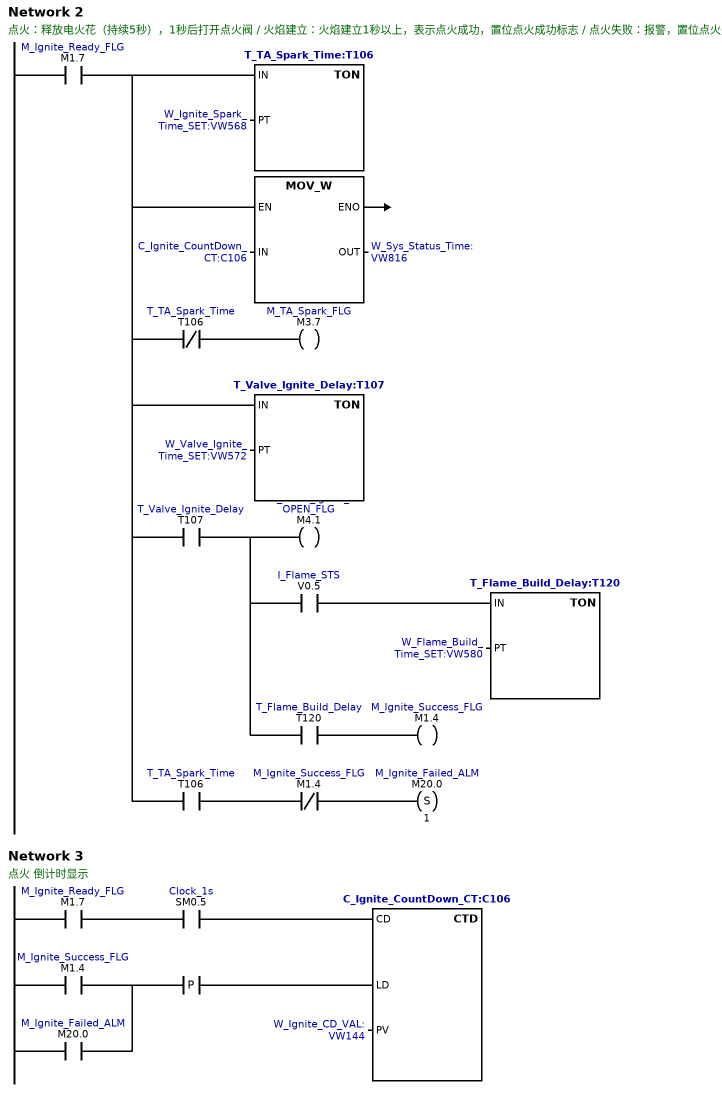
Network 2
// 点火：释放电火花（持续5秒），1秒后打开点火阀
// 火焰建立：火焰建立1秒以上，表示点火成功，置位点火成功标志
// 点火失败：报警，置位点火失败报警信号
// 
// 
// 
LD     M_Ignite_Ready_FLG:M1.7
LPS
TON    T_TA_Spark_Time:T106, W_Ignite_Spark_Time_SET:VW568
MOVW   C_Ignite_CountDown_CT:C106, W_Sys_Status_Time:VW816
AN     T_TA_Spark_Time:T106
=      M_TA_Spark_FLG:M3.7
LRD
TON    T_Valve_Ignite_Delay:T107, W_Valve_Ignite_Time_SET:VW572
LRD
A      T_Valve_Ignite_Delay:T107
LPS
=      M_Valve_Ignite_OPEN_FLG:M4.1
A      I_Flame_STS:V0.5
TON    T_Flame_Build_Delay:T120, W_Flame_Build_Time_SET:VW580
LPP
A      T_Flame_Build_Delay:T120
=      M_Ignite_Success_FLG:M1.4
LPP
A      T_TA_Spark_Time:T106
AN     M_Ignite_Success_FLG:M1.4
S      M_Ignite_Failed_ALM:M20.0, 1
Network 3
// 点火 倒计时显示
LD     M_Ignite_Ready_FLG:M1.7
A      Clock_1s:SM0.5
LD     M_Ignite_Success_FLG:M1.4
O      M_Ignite_Failed_ALM:M20.0
EU
CTD    C_Ignite_CountDown_CT:C106, W_Ignite_CD_VAL:VW144
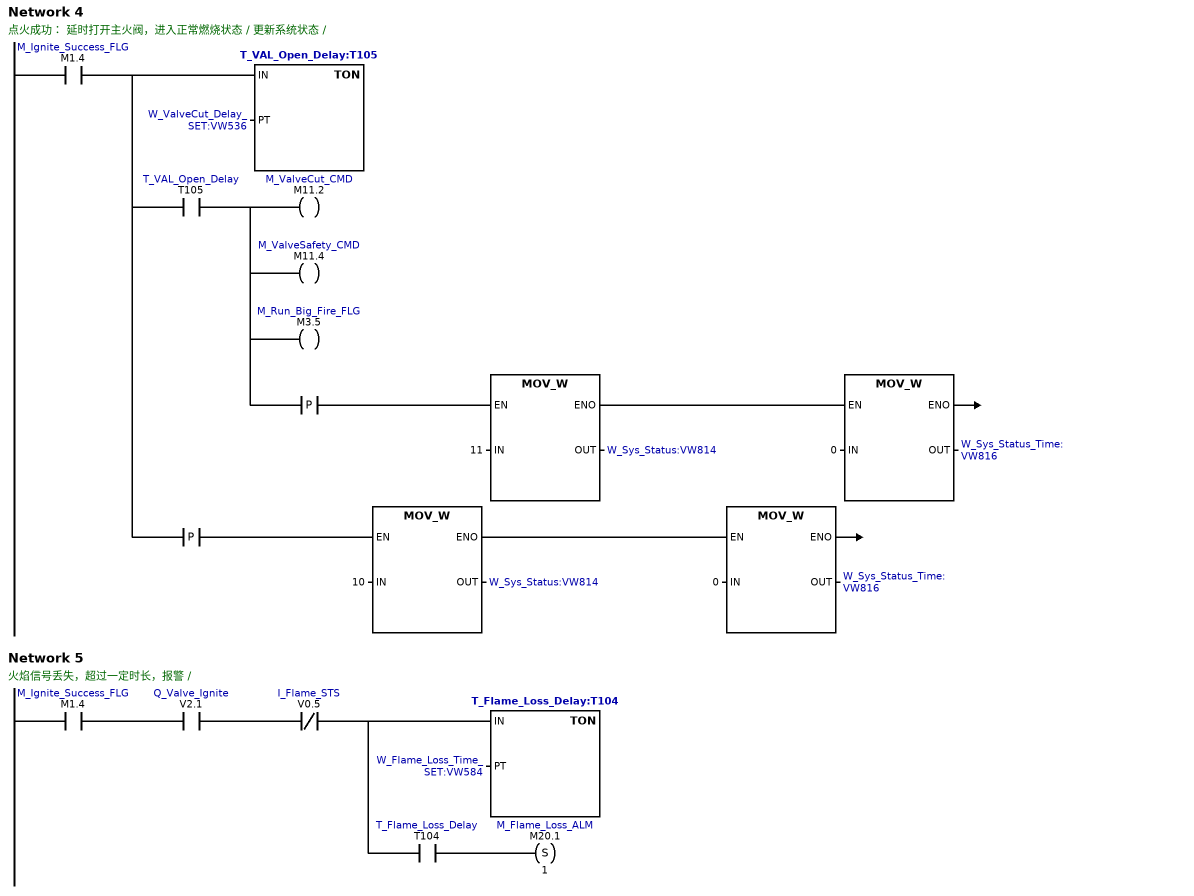
Network 4
// 点火成功： 延时打开主火阀，进入正常燃烧状态
// 更新系统状态
// 
LD     M_Ignite_Success_FLG:M1.4
LPS
TON    T_VAL_Open_Delay:T105, W_ValveCut_Delay_SET:VW536
A      T_VAL_Open_Delay:T105
=      M_ValveCut_CMD:M11.2
=      M_ValveSafety_CMD:M11.4
=      M_Run_Big_Fire_FLG:M3.5
EU
MOVW   11, W_Sys_Status:VW814
AENO
MOVW   0, W_Sys_Status_Time:VW816
LPP
EU
MOVW   10, W_Sys_Status:VW814
AENO
MOVW   0, W_Sys_Status_Time:VW816
Network 5
// 火焰信号丢失，超过一定时长，报警
// 
LD     M_Ignite_Success_FLG:M1.4
A      Q_Valve_Ignite:V2.1
AN     I_Flame_STS:V0.5
TON    T_Flame_Loss_Delay:T104, W_Flame_Loss_Time_SET:VW584
A      T_Flame_Loss_Delay:T104
S      M_Flame_Loss_ALM:M20.1, 1
Network 6
// 超温停机,
// 1、当前温度大于停机温度超过3秒停主火，
// 2、温度低于开机温度超过3秒，开主火；
END_SUBROUTINE_BLOCK

SUBROUTINE_BLOCK 阶段升温:SBR5
TITLE=
BEGIN
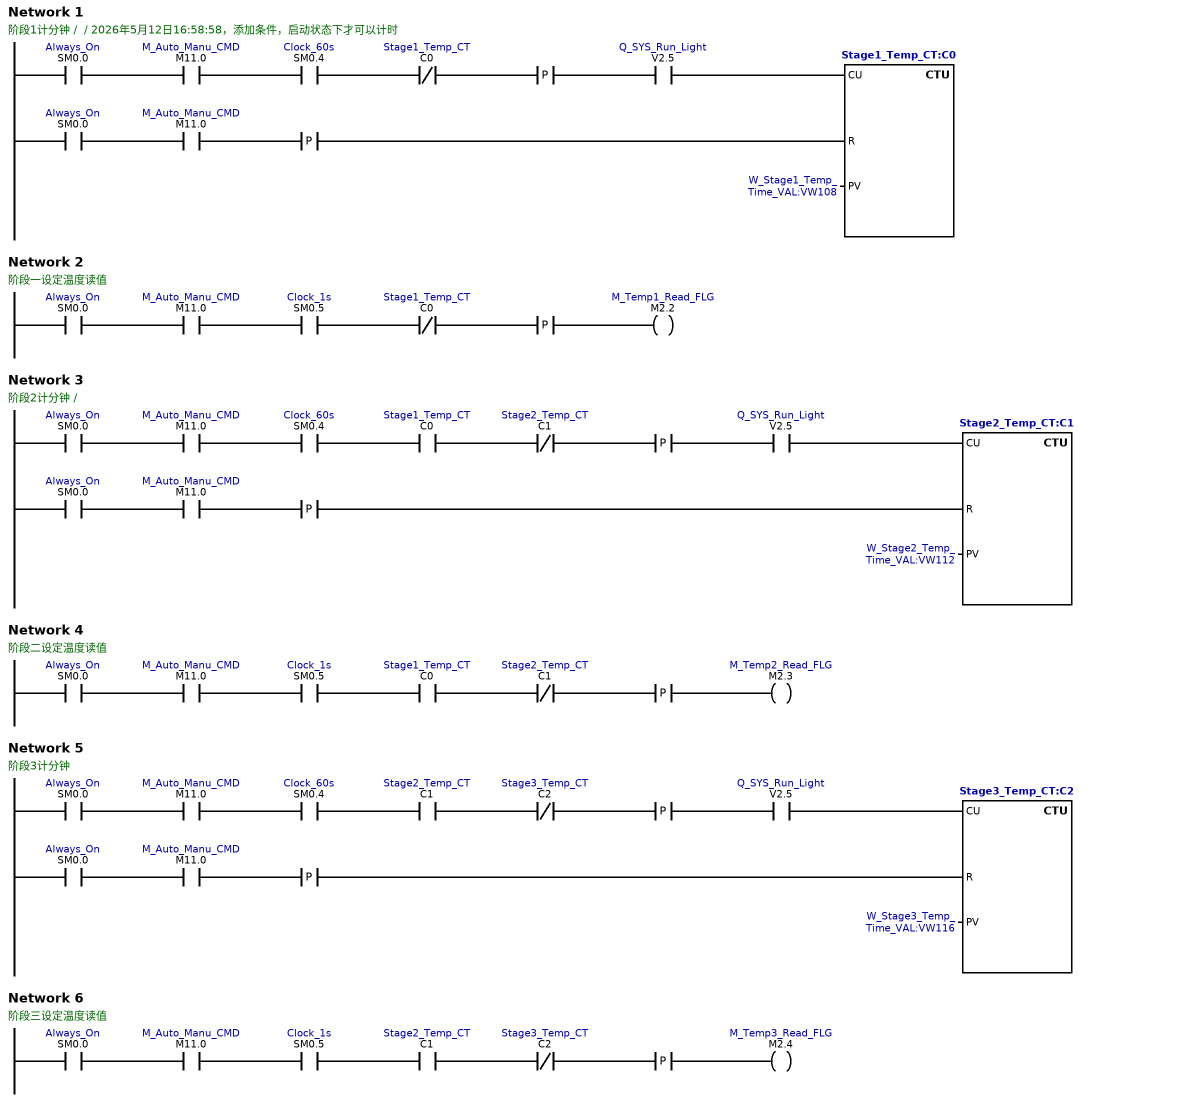
Network 1
// 阶段1计分钟
// 
// 2026年5月12日16:58:58，添加条件，启动状态下才可以计时
LD     Always_On:SM0.0
A      M_Auto_Manu_CMD:M11.0
A      Clock_60s:SM0.4
AN     Stage1_Temp_CT:C0
EU
A      Q_SYS_Run_Light:V2.5
LD     Always_On:SM0.0
A      M_Auto_Manu_CMD:M11.0
EU
CTU    Stage1_Temp_CT:C0, W_Stage1_Temp_Time_VAL:VW108
Network 2
// 阶段一设定温度读值
LD     Always_On:SM0.0
A      M_Auto_Manu_CMD:M11.0
A      Clock_1s:SM0.5
AN     Stage1_Temp_CT:C0
EU
=      M_Temp1_Read_FLG:M2.2
Network 3
// 阶段2计分钟
// 
LD     Always_On:SM0.0
A      M_Auto_Manu_CMD:M11.0
A      Clock_60s:SM0.4
A      Stage1_Temp_CT:C0
AN     Stage2_Temp_CT:C1
EU
A      Q_SYS_Run_Light:V2.5
LD     Always_On:SM0.0
A      M_Auto_Manu_CMD:M11.0
EU
CTU    Stage2_Temp_CT:C1, W_Stage2_Temp_Time_VAL:VW112
Network 4
// 阶段二设定温度读值
LD     Always_On:SM0.0
A      M_Auto_Manu_CMD:M11.0
A      Clock_1s:SM0.5
A      Stage1_Temp_CT:C0
AN     Stage2_Temp_CT:C1
EU
=      M_Temp2_Read_FLG:M2.3
Network 5
// 阶段3计分钟
LD     Always_On:SM0.0
A      M_Auto_Manu_CMD:M11.0
A      Clock_60s:SM0.4
A      Stage2_Temp_CT:C1
AN     Stage3_Temp_CT:C2
EU
A      Q_SYS_Run_Light:V2.5
LD     Always_On:SM0.0
A      M_Auto_Manu_CMD:M11.0
EU
CTU    Stage3_Temp_CT:C2, W_Stage3_Temp_Time_VAL:VW116
Network 6
// 阶段三设定温度读值
LD     Always_On:SM0.0
A      M_Auto_Manu_CMD:M11.0
A      Clock_1s:SM0.5
A      Stage2_Temp_CT:C1
AN     Stage3_Temp_CT:C2
EU
=      M_Temp3_Read_FLG:M2.4
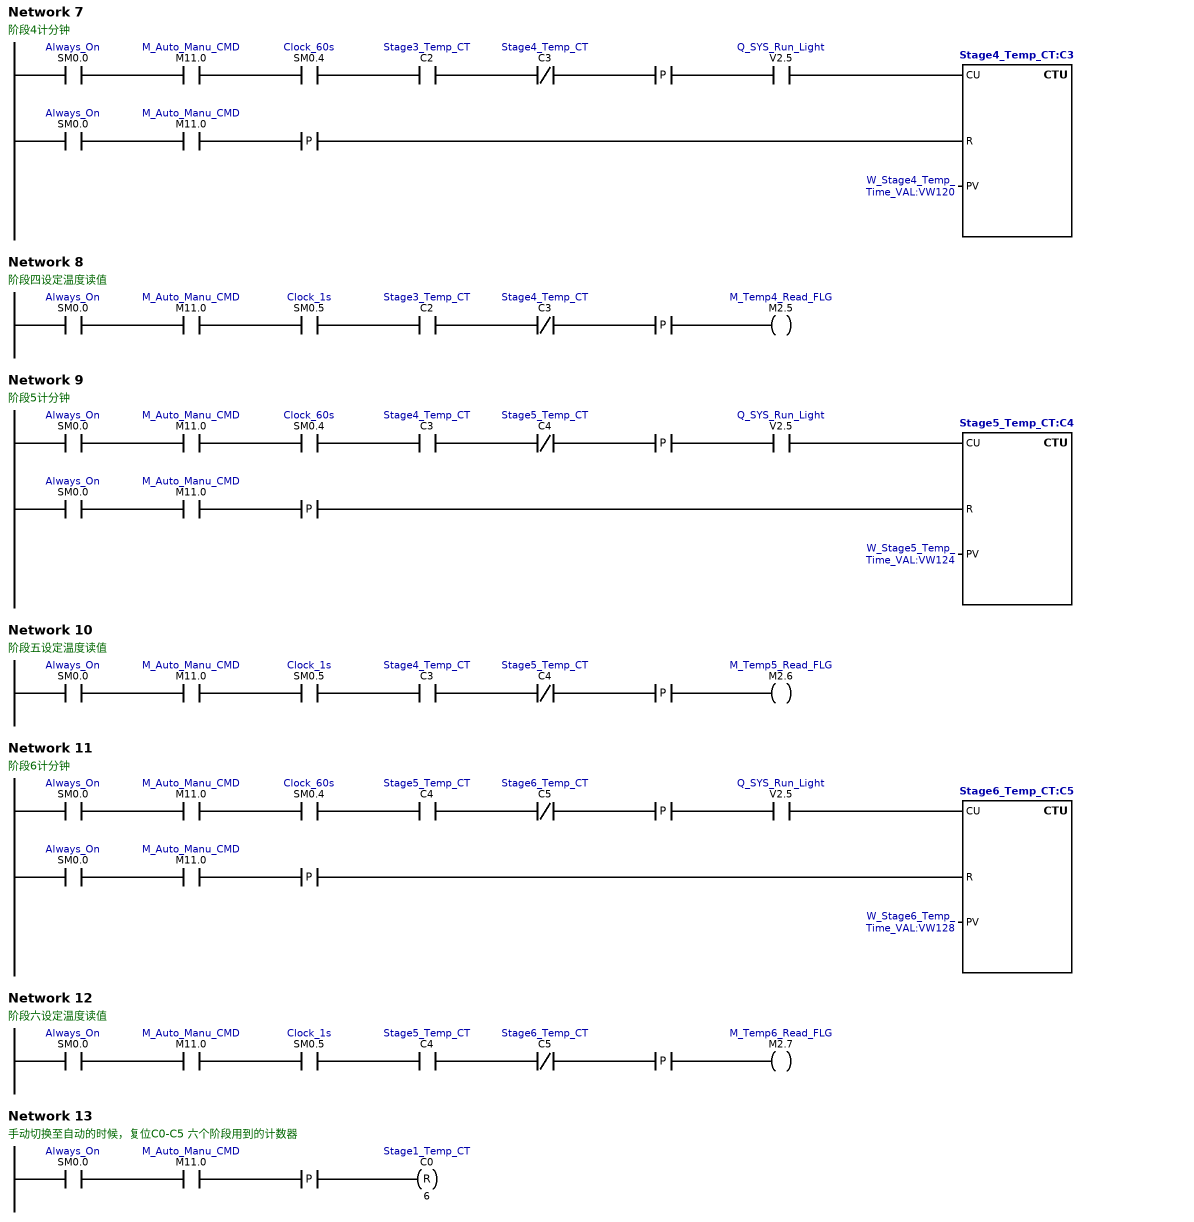
Network 7
// 阶段4计分钟
LD     Always_On:SM0.0
A      M_Auto_Manu_CMD:M11.0
A      Clock_60s:SM0.4
A      Stage3_Temp_CT:C2
AN     Stage4_Temp_CT:C3
EU
A      Q_SYS_Run_Light:V2.5
LD     Always_On:SM0.0
A      M_Auto_Manu_CMD:M11.0
EU
CTU    Stage4_Temp_CT:C3, W_Stage4_Temp_Time_VAL:VW120
Network 8
// 阶段四设定温度读值
LD     Always_On:SM0.0
A      M_Auto_Manu_CMD:M11.0
A      Clock_1s:SM0.5
A      Stage3_Temp_CT:C2
AN     Stage4_Temp_CT:C3
EU
=      M_Temp4_Read_FLG:M2.5
Network 9
// 阶段5计分钟
LD     Always_On:SM0.0
A      M_Auto_Manu_CMD:M11.0
A      Clock_60s:SM0.4
A      Stage4_Temp_CT:C3
AN     Stage5_Temp_CT:C4
EU
A      Q_SYS_Run_Light:V2.5
LD     Always_On:SM0.0
A      M_Auto_Manu_CMD:M11.0
EU
CTU    Stage5_Temp_CT:C4, W_Stage5_Temp_Time_VAL:VW124
Network 10
// 阶段五设定温度读值
LD     Always_On:SM0.0
A      M_Auto_Manu_CMD:M11.0
A      Clock_1s:SM0.5
A      Stage4_Temp_CT:C3
AN     Stage5_Temp_CT:C4
EU
=      M_Temp5_Read_FLG:M2.6
Network 11
// 阶段6计分钟
LD     Always_On:SM0.0
A      M_Auto_Manu_CMD:M11.0
A      Clock_60s:SM0.4
A      Stage5_Temp_CT:C4
AN     Stage6_Temp_CT:C5
EU
A      Q_SYS_Run_Light:V2.5
LD     Always_On:SM0.0
A      M_Auto_Manu_CMD:M11.0
EU
CTU    Stage6_Temp_CT:C5, W_Stage6_Temp_Time_VAL:VW128
Network 12
// 阶段六设定温度读值
LD     Always_On:SM0.0
A      M_Auto_Manu_CMD:M11.0
A      Clock_1s:SM0.5
A      Stage5_Temp_CT:C4
AN     Stage6_Temp_CT:C5
EU
=      M_Temp6_Read_FLG:M2.7
Network 13
// 手动切换至自动的时候，复位C0-C5 六个阶段用到的计数器
LD     Always_On:SM0.0
A      M_Auto_Manu_CMD:M11.0
EU
R      Stage1_Temp_CT:C0, 6
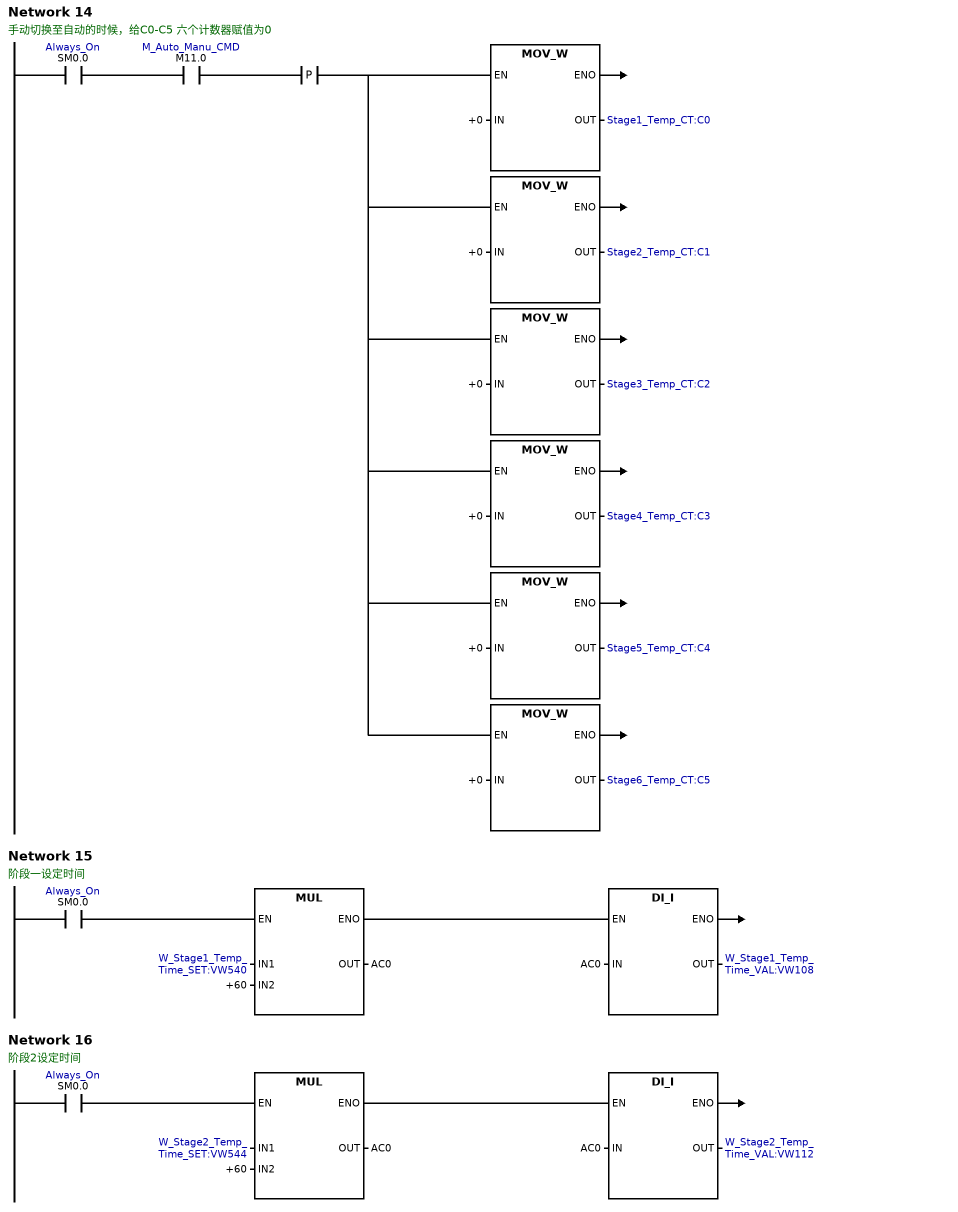
Network 14
// 手动切换至自动的时候，给C0-C5 六个计数器赋值为0
LD     Always_On:SM0.0
A      M_Auto_Manu_CMD:M11.0
EU
MOVW   +0, Stage1_Temp_CT:C0
MOVW   +0, Stage2_Temp_CT:C1
MOVW   +0, Stage3_Temp_CT:C2
MOVW   +0, Stage4_Temp_CT:C3
MOVW   +0, Stage5_Temp_CT:C4
MOVW   +0, Stage6_Temp_CT:C5
Network 15
// 阶段一设定时间
LD     Always_On:SM0.0
MOVW   W_Stage1_Temp_Time_SET:VW540, AC0
AENO
MUL    +60, AC0
AENO
DTI    AC0, W_Stage1_Temp_Time_VAL:VW108
Network 16
// 阶段2设定时间
LD     Always_On:SM0.0
MOVW   W_Stage2_Temp_Time_SET:VW544, AC0
AENO
MUL    +60, AC0
AENO
DTI    AC0, W_Stage2_Temp_Time_VAL:VW112
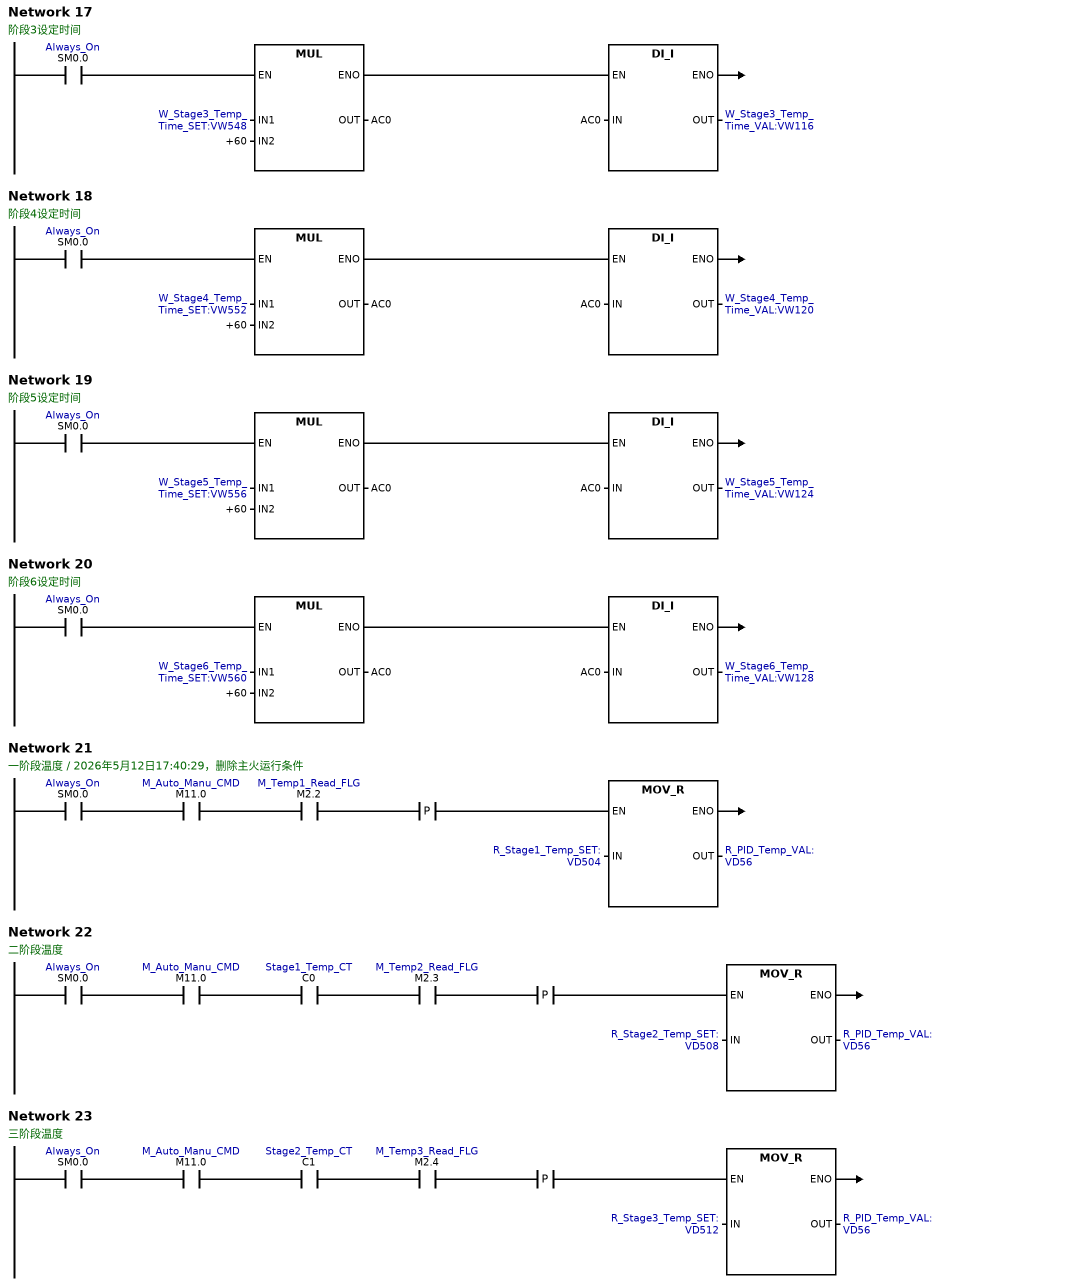
Network 17
// 阶段3设定时间
LD     Always_On:SM0.0
MOVW   W_Stage3_Temp_Time_SET:VW548, AC0
AENO
MUL    +60, AC0
AENO
DTI    AC0, W_Stage3_Temp_Time_VAL:VW116
Network 18
// 阶段4设定时间
LD     Always_On:SM0.0
MOVW   W_Stage4_Temp_Time_SET:VW552, AC0
AENO
MUL    +60, AC0
AENO
DTI    AC0, W_Stage4_Temp_Time_VAL:VW120
Network 19
// 阶段5设定时间
LD     Always_On:SM0.0
MOVW   W_Stage5_Temp_Time_SET:VW556, AC0
AENO
MUL    +60, AC0
AENO
DTI    AC0, W_Stage5_Temp_Time_VAL:VW124
Network 20
// 阶段6设定时间
LD     Always_On:SM0.0
MOVW   W_Stage6_Temp_Time_SET:VW560, AC0
AENO
MUL    +60, AC0
AENO
DTI    AC0, W_Stage6_Temp_Time_VAL:VW128
Network 21
// 一阶段温度
// 2026年5月12日17:40:29，删除主火运行条件
LD     Always_On:SM0.0
A      M_Auto_Manu_CMD:M11.0
A      M_Temp1_Read_FLG:M2.2
EU
MOVR   R_Stage1_Temp_SET:VD504, R_PID_Temp_VAL:VD56
Network 22
// 二阶段温度
LD     Always_On:SM0.0
A      M_Auto_Manu_CMD:M11.0
A      Stage1_Temp_CT:C0
A      M_Temp2_Read_FLG:M2.3
EU
MOVR   R_Stage2_Temp_SET:VD508, R_PID_Temp_VAL:VD56
Network 23
// 三阶段温度
LD     Always_On:SM0.0
A      M_Auto_Manu_CMD:M11.0
A      Stage2_Temp_CT:C1
A      M_Temp3_Read_FLG:M2.4
EU
MOVR   R_Stage3_Temp_SET:VD512, R_PID_Temp_VAL:VD56
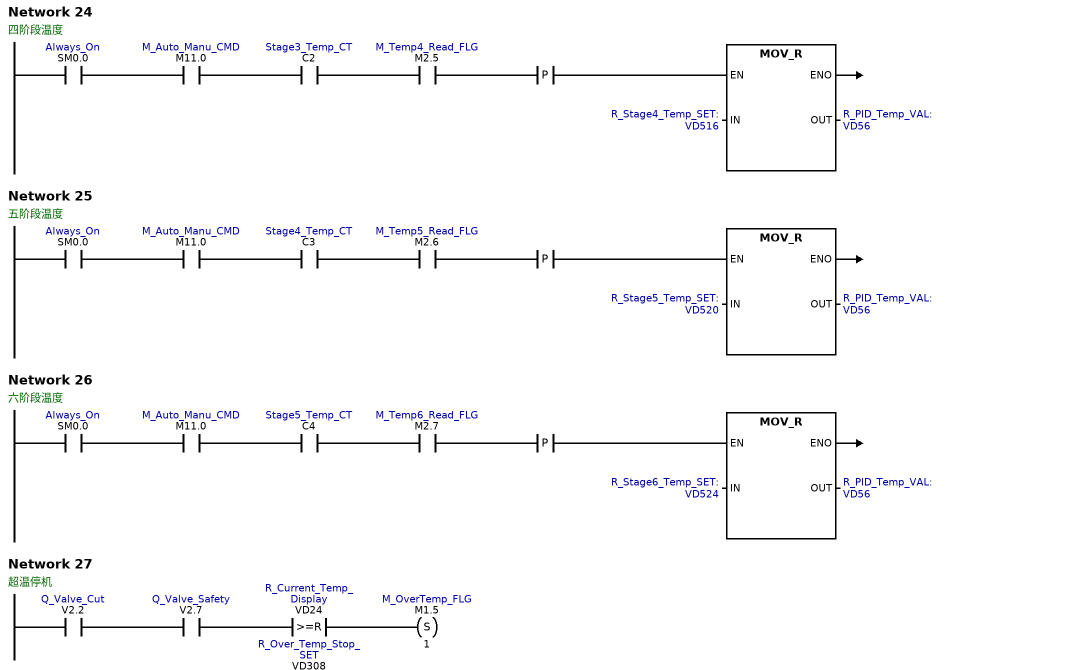
Network 24
// 四阶段温度
LD     Always_On:SM0.0
A      M_Auto_Manu_CMD:M11.0
A      Stage3_Temp_CT:C2
A      M_Temp4_Read_FLG:M2.5
EU
MOVR   R_Stage4_Temp_SET:VD516, R_PID_Temp_VAL:VD56
Network 25
// 五阶段温度
LD     Always_On:SM0.0
A      M_Auto_Manu_CMD:M11.0
A      Stage4_Temp_CT:C3
A      M_Temp5_Read_FLG:M2.6
EU
MOVR   R_Stage5_Temp_SET:VD520, R_PID_Temp_VAL:VD56
Network 26
// 六阶段温度
LD     Always_On:SM0.0
A      M_Auto_Manu_CMD:M11.0
A      Stage5_Temp_CT:C4
A      M_Temp6_Read_FLG:M2.7
EU
MOVR   R_Stage6_Temp_SET:VD524, R_PID_Temp_VAL:VD56
Network 27
// 超温停机
LD     Q_Valve_Cut:V2.2
A      Q_Valve_Safety:V2.7
AR>=   R_Current_Temp_Display:VD24, R_Over_Temp_Stop_SET:VD308
S      M_OverTemp_FLG:M1.5, 1
END_SUBROUTINE_BLOCK

SUBROUTINE_BLOCK 开度档位:SBR6
TITLE=开度档位子程序
// 功能：
// 1、处理每档对应的燃气调节阀开度多少，空气调节阀开度多少。
// 2、手动模式，升档、降档控制
// 3、自动模式，PID输出转换成档位处理
// 
BEGIN
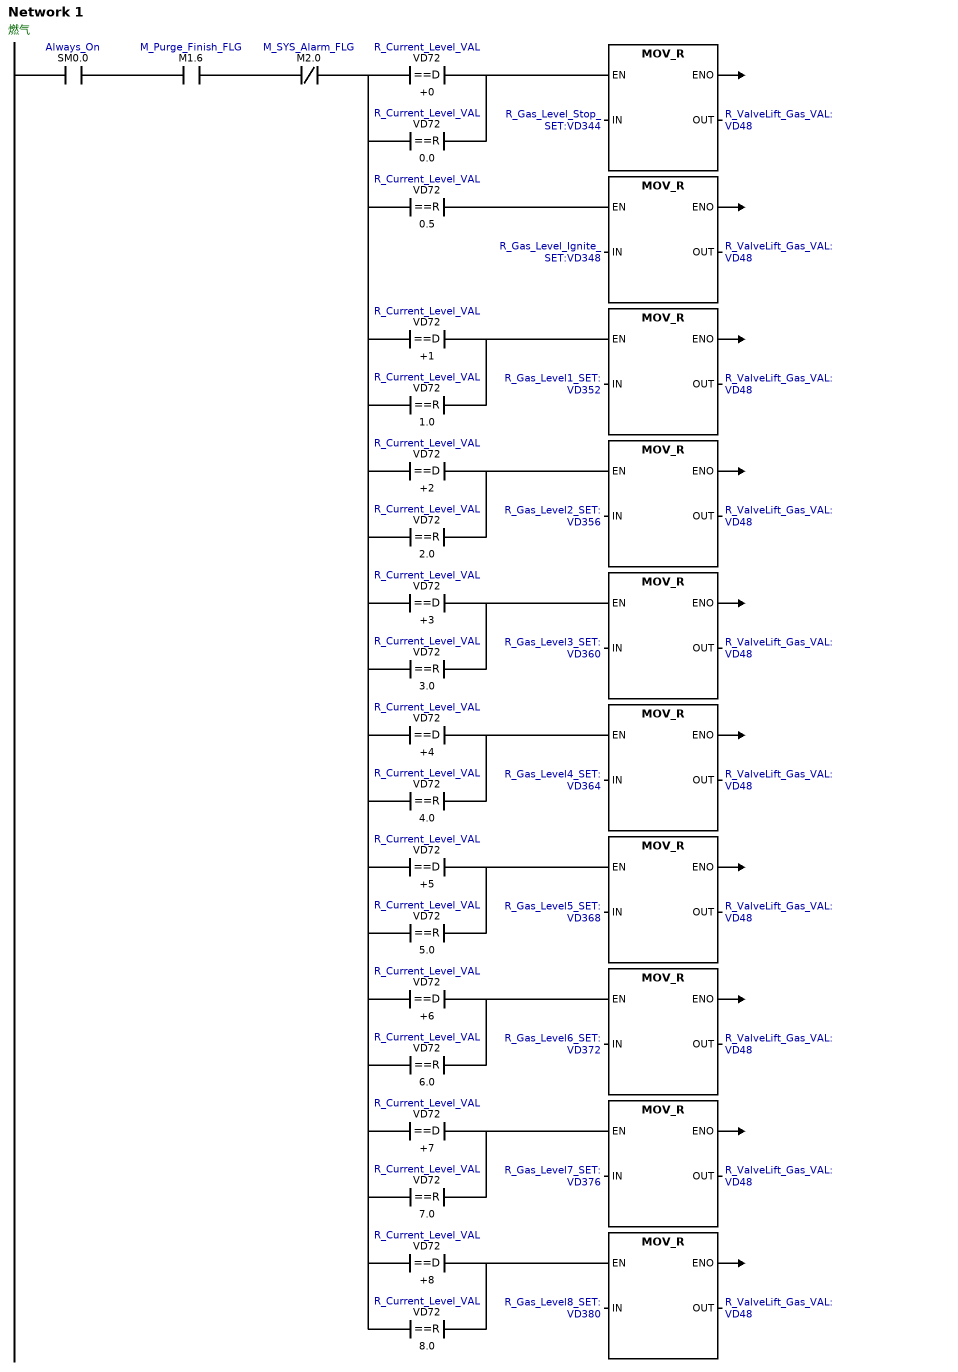
Network 1
// 燃气
LD     Always_On:SM0.0
A      M_Purge_Finish_FLG:M1.6
AN     M_SYS_Alarm_FLG:M2.0
LPS
LDD=   R_Current_Level_VAL:VD72, +0
OR=    R_Current_Level_VAL:VD72, 0.0
ALD
MOVR   R_Gas_Level_Stop_SET:VD344, R_ValveLift_Gas_VAL:VD48
LRD
AR=    R_Current_Level_VAL:VD72, 0.5
MOVR   R_Gas_Level_Ignite_SET:VD348, R_ValveLift_Gas_VAL:VD48
LRD
LDD=   R_Current_Level_VAL:VD72, +1
OR=    R_Current_Level_VAL:VD72, 1.0
ALD
MOVR   R_Gas_Level1_SET:VD352, R_ValveLift_Gas_VAL:VD48
LRD
LDD=   R_Current_Level_VAL:VD72, +2
OR=    R_Current_Level_VAL:VD72, 2.0
ALD
MOVR   R_Gas_Level2_SET:VD356, R_ValveLift_Gas_VAL:VD48
LRD
LDD=   R_Current_Level_VAL:VD72, +3
OR=    R_Current_Level_VAL:VD72, 3.0
ALD
MOVR   R_Gas_Level3_SET:VD360, R_ValveLift_Gas_VAL:VD48
LRD
LDD=   R_Current_Level_VAL:VD72, +4
OR=    R_Current_Level_VAL:VD72, 4.0
ALD
MOVR   R_Gas_Level4_SET:VD364, R_ValveLift_Gas_VAL:VD48
LRD
LDD=   R_Current_Level_VAL:VD72, +5
OR=    R_Current_Level_VAL:VD72, 5.0
ALD
MOVR   R_Gas_Level5_SET:VD368, R_ValveLift_Gas_VAL:VD48
LRD
LDD=   R_Current_Level_VAL:VD72, +6
OR=    R_Current_Level_VAL:VD72, 6.0
ALD
MOVR   R_Gas_Level6_SET:VD372, R_ValveLift_Gas_VAL:VD48
LRD
LDD=   R_Current_Level_VAL:VD72, +7
OR=    R_Current_Level_VAL:VD72, 7.0
ALD
MOVR   R_Gas_Level7_SET:VD376, R_ValveLift_Gas_VAL:VD48
LPP
LDD=   R_Current_Level_VAL:VD72, +8
OR=    R_Current_Level_VAL:VD72, 8.0
ALD
MOVR   R_Gas_Level8_SET:VD380, R_ValveLift_Gas_VAL:VD48
